LIN {X 0.159,Y -655.159,Z 842.614,A 0.000,B 0.000,C 90.000,E1 326.580} C_DIS
LIN {X 0.166,Y -657.931,Z 842.609,A 0.000,B 0.000,C 90.000,E1 325.595} C_DIS
LIN {X 0.218,Y -660.579,Z 842.604,A 0.000,B 0.000,C 90.000,E1 324.609} C_DIS
LIN {X -0.133,Y -663.447,Z 842.597,A 0.000,B 0.000,C 90.000,E1 323.417} C_DIS
LIN {X -0.112,Y -664.973,Z 842.593,A 0.000,B 0.000,C 90.000,E1 322.683} C_DIS
LIN {X 0.021,Y -666.876,Z 842.587,A 0.000,B 0.000,C 90.000,E1 321.698} C_DIS
LIN {X 0.058,Y -668.914,Z 842.581,A 0.000,B 0.000,C 90.000,E1 320.481} C_DIS
LIN {X -0.293,Y -670.706,Z 842.574,A 0.000,B 0.000,C 90.000,E1 319.299} C_DIS
LIN {X 0.364,Y -673.373,Z 842.563,A 0.000,B 0.000,C 90.000,E1 317.310} C_DIS
LIN {X -0.033,Y -674.352,Z 842.559,A 0.000,B 0.000,C 90.000,E1 316.620} C_DIS
LIN {X 0.016,Y -675.024,Z 842.556,A 0.000,B 0.000,C 90.000,E1 316.134} C_DIS
LIN {X 0.071,Y -675.502,Z 842.554,A 0.000,B 0.000,C 90.000,E1 315.648} C_DIS
LIN {X 0.131,Y -676.141,Z 842.551,A 0.000,B 0.000,C 90.000,E1 315.162} C_DIS
LIN {X 0.331,Y -677.702,Z 842.543,A 0.000,B 0.000,C 90.000,E1 313.704} C_DIS
LIN {X 0.049,Y -678.975,Z 842.536,A 0.000,B 0.000,C 90.000,E1 312.528} C_DIS
LIN {X 0.331,Y -680.489,Z 842.528,A 0.000,B 0.000,C 90.000,E1 311.067} C_DIS
LIN {X 0.196,Y -681.842,Z 842.520,A 0.000,B 0.000,C 90.000,E1 309.644} C_DIS
LIN {X -0.311,Y -683.305,Z 842.511,A 0.000,B 0.000,C 90.000,E1 308.016} C_DIS
LIN {X -0.286,Y -684.517,Z 842.503,A 0.000,B 0.000,C 90.000,E1 306.583} C_DIS
LIN {X 0.318,Y -685.661,Z 842.495,A 0.000,B 0.000,C 90.000,E1 305.105} C_DIS
LIN {X 0.359,Y -686.472,Z 842.489,A 0.000,B 0.000,C 90.000,E1 303.913} C_DIS
LIN {X -0.135,Y -687.817,Z 842.478,A 0.000,B 0.000,C 90.000,E1 302.054} C_DIS
LIN {X 0.207,Y -689.207,Z 842.468,A 0.000,B 0.000,C 90.000,E1 300.129} C_DIS
LIN {X 0.017,Y -690.515,Z 842.458,A 0.000,B 0.000,C 90.000,E1 298.487} C_DIS
LIN {X -0.095,Y -691.710,Z 842.450,A 0.000,B 0.000,C 90.000,E1 297.078} C_DIS
LIN {X 0.068,Y -693.228,Z 842.441,A 0.000,B 0.000,C 90.000,E1 295.412} C_DIS
LIN {X 0.137,Y -694.043,Z 842.436,A 0.000,B 0.000,C 90.000,E1 294.463} C_DIS
LIN {X -0.037,Y -694.284,Z 842.432,A 0.000,B 0.000,C 90.000,E1 293.770} C_DIS
LIN {X 0.182,Y -693.984,Z 842.430,A 0.000,B 0.000,C 90.000,E1 293.281} C_DIS
LIN {X -0.211,Y -693.555,Z 842.428,A 0.000,B 0.000,C 90.000,E1 293.078} C_DIS
LIN {X 0.125,Y -691.002,Z 842.425,A 0.000,B 0.000,C 90.000,E1 292.461} C_DIS
LIN {X 0.242,Y -690.176,Z 842.424,A 0.000,B 0.000,C 90.000,E1 292.333} C_DIS
LIN {X 0.358,Y -688.960,Z 842.424,A 0.000,B 0.000,C 90.000,E1 292.206} C_DIS
LIN {X -0.397,Y -683.079,Z 842.421,A 0.000,B 0.000,C 90.000,E1 291.844} C_DIS
LIN {X -0.059,Y -681.119,Z 842.421,A 0.000,B 0.000,C 90.000,E1 291.716} C_DIS
LIN {X -0.296,Y -671.354,Z 842.419,A 0.000,B 0.000,C 90.000,E1 291.408} C_DIS
LIN {X 0.171,Y -664.788,Z 842.418,A 0.000,B 0.000,C 90.000,E1 291.227} C_DIS
LIN {X -0.028,Y -654.109,Z 842.417,A 0.000,B 0.000,C 90.000,E1 291.046} C_DIS
LIN {X -0.109,Y -648.329,Z 842.416,A 0.000,B 0.000,C 90.000,E1 290.918} C_DIS
LIN {X -0.062,Y -642.259,Z 842.415,A 0.000,B 0.000,C 90.000,E1 290.737} C_DIS
LIN {X -0.135,Y -636.875,Z 842.414,A 0.000,B 0.000,C 90.000,E1 290.536} C_DIS
LIN {X -0.105,Y -634.934,Z 842.414,A 0.000,B 0.000,C 90.000,E1 290.429} C_DIS
LIN {X -0.127,Y -632.025,Z 842.412,A 0.000,B 0.000,C 90.000,E1 290.248} C_DIS
LIN {X -0.160,Y -631.973,Z 842.412,A 0.000,B 0.000,C 90.000,E1 290.248} C_DIS
LIN {X -0.137,Y -631.192,Z 842.412,A 0.000,B 0.000,C 90.000,E1 290.120} C_DIS
LIN {X -0.180,Y -631.170,Z 842.412,A 0.000,B 0.000,C 90.000,E1 290.120} C_DIS
LIN {X -0.162,Y -631.443,Z 842.410,A 0.000,B 0.000,C 90.000,E1 289.885} C_DIS
LIN {X -0.156,Y -631.746,Z 842.410,A 0.000,B 0.000,C 90.000,E1 289.758} C_DIS
LIN {X 0.257,Y -633.950,Z 842.407,A 0.000,B 0.000,C 90.000,E1 289.214} C_DIS
LIN {X -0.086,Y -638.971,Z 842.402,A 0.000,B 0.000,C 90.000,E1 288.362} C_DIS
LIN {X -0.231,Y -641.589,Z 842.399,A 0.000,B 0.000,C 90.000,E1 287.873} C_DIS
LIN {X 0.090,Y -644.996,Z 842.395,A 0.000,B 0.000,C 90.000,E1 287.094} C_DIS
LIN {X -0.211,Y -647.076,Z 842.392,A 0.000,B 0.000,C 90.000,E1 286.622} C_DIS
LIN {X 0.168,Y -649.848,Z 842.388,A 0.000,B 0.000,C 90.000,E1 285.843} C_DIS
LIN {X -0.228,Y -652.100,Z 842.384,A 0.000,B 0.000,C 90.000,E1 285.134} C_DIS
LIN {X 0.319,Y -653.323,Z 842.381,A 0.000,B 0.000,C 90.000,E1 284.592} C_DIS
LIN {X -0.044,Y -654.775,Z 842.377,A 0.000,B 0.000,C 90.000,E1 283.883} C_DIS
LIN {X -0.278,Y -655.578,Z 842.374,A 0.000,B 0.000,C 90.000,E1 283.411} C_DIS
LIN {X 0.017,Y -656.130,Z 842.370,A 0.000,B 0.000,C 90.000,E1 282.647} C_DIS
LIN {X -0.211,Y -656.299,Z 842.368,A 0.000,B 0.000,C 90.000,E1 282.175} C_DIS
LIN {X 0.070,Y -656.221,Z 842.365,A 0.000,B 0.000,C 90.000,E1 281.658} C_DIS
LIN {X -0.158,Y -655.977,Z 842.362,A 0.000,B 0.000,C 90.000,E1 281.186} C_DIS
LIN {X 0.016,Y -655.114,Z 842.358,A 0.000,B 0.000,C 90.000,E1 280.433} C_DIS
LIN {X -0.222,Y -654.223,Z 842.355,A 0.000,B 0.000,C 90.000,E1 279.962} C_DIS
LIN {X 0.064,Y -653.145,Z 842.353,A 0.000,B 0.000,C 90.000,E1 279.443} C_DIS
LIN {X -0.193,Y -651.664,Z 842.350,A 0.000,B 0.000,C 90.000,E1 278.973} C_DIS
LIN {X 0.080,Y -649.679,Z 842.347,A 0.000,B 0.000,C 90.000,E1 278.454} C_DIS
LIN {X 0.312,Y -646.763,Z 842.344,A 0.000,B 0.000,C 90.000,E1 277.814} C_DIS
LIN {X -0.210,Y -643.271,Z 842.340,A 0.000,B 0.000,C 90.000,E1 277.239} C_DIS
LIN {X 0.133,Y -640.882,Z 842.338,A 0.000,B 0.000,C 90.000,E1 276.834} C_DIS
LIN {X -0.119,Y -638.988,Z 842.337,A 0.000,B 0.000,C 90.000,E1 276.606} C_DIS
LIN {X 0.072,Y -634.956,Z 842.334,A 0.000,B 0.000,C 90.000,E1 276.087} C_DIS
LIN {X -0.092,Y -631.561,Z 842.332,A 0.000,B 0.000,C 90.000,E1 275.739} C_DIS
LIN {X -0.193,Y -630.344,Z 842.331,A 0.000,B 0.000,C 90.000,E1 275.625} C_DIS
LIN {X -0.178,Y -625.082,Z 842.329,A 0.000,B 0.000,C 90.000,E1 275.163} C_DIS
LIN {X -0.078,Y -623.753,Z 842.328,A 0.000,B 0.000,C 90.000,E1 275.049} C_DIS
LIN {X -0.272,Y -617.463,Z 842.326,A 0.000,B 0.000,C 90.000,E1 274.645} C_DIS
LIN {X -0.035,Y -611.108,Z 842.324,A 0.000,B 0.000,C 90.000,E1 274.245} C_DIS
LIN {X 0.029,Y -604.288,Z 842.322,A 0.000,B 0.000,C 90.000,E1 273.898} C_DIS
LIN {X -0.269,Y -597.399,Z 842.320,A 0.000,B 0.000,C 90.000,E1 273.612} C_DIS
LIN {X -0.131,Y -591.984,Z 842.319,A 0.000,B 0.000,C 90.000,E1 273.383} C_DIS
LIN {X 0.225,Y -584.869,Z 842.317,A 0.000,B 0.000,C 90.000,E1 273.094} C_DIS
LIN {X -0.174,Y -578.917,Z 842.317,A 0.000,B 0.000,C 90.000,E1 272.980} C_DIS
LIN {X -0.269,Y -572.255,Z 842.316,A 0.000,B 0.000,C 90.000,E1 272.865} C_DIS
LIN {X 0.167,Y -564.435,Z 842.315,A 0.000,B 0.000,C 90.000,E1 272.751} C_DIS
LIN {X 0.112,Y -560.003,Z 842.315,A 0.000,B 0.000,C 90.000,E1 272.751} C_DIS
LIN {X -0.196,Y -554.623,Z 842.315,A 0.000,B 0.000,C 90.000,E1 272.751} C_DIS
LIN {X 0.215,Y -553.395,Z 842.315,A 0.000,B 0.000,C 90.000,E1 272.694} C_DIS
LIN {X 0.227,Y -550.457,Z 842.315,A 0.000,B 0.000,C 90.000,E1 272.579} C_DIS
LIN {X 0.187,Y -550.405,Z 842.315,A 0.000,B 0.000,C 90.000,E1 272.579} C_DIS
LIN {X 0.172,Y -549.400,Z 842.314,A 0.000,B 0.000,C 90.000,E1 272.407} C_DIS
LIN {X 0.209,Y -548.528,Z 842.312,A 0.000,B 0.000,C 90.000,E1 272.121} C_DIS
LIN {X -0.222,Y -547.535,Z 842.309,A 0.000,B 0.000,C 90.000,E1 271.604} C_DIS
LIN {X 0.004,Y -546.052,Z 842.301,A 0.000,B 0.000,C 90.000,E1 270.172} C_DIS
LIN {X -0.267,Y -544.563,Z 842.290,A 0.000,B 0.000,C 90.000,E1 268.224} C_DIS
LIN {X -0.055,Y -543.574,Z 842.282,A 0.000,B 0.000,C 90.000,E1 266.788} C_DIS
LIN {X 0.111,Y -542.607,Z 842.274,A 0.000,B 0.000,C 90.000,E1 265.355} C_DIS
LIN {X -0.193,Y -541.693,Z 842.266,A 0.000,B 0.000,C 90.000,E1 263.970} C_DIS
LIN {X -0.105,Y -541.008,Z 842.262,A 0.000,B 0.000,C 90.000,E1 263.109} C_DIS
LIN {X 0.165,Y -539.463,Z 842.252,A 0.000,B 0.000,C 90.000,E1 261.376} C_DIS
LIN {X -0.116,Y -538.157,Z 842.244,A 0.000,B 0.000,C 90.000,E1 259.982} C_DIS
LIN {X -0.196,Y -536.114,Z 842.233,A 0.000,B 0.000,C 90.000,E1 257.993} C_DIS
LIN {X 0.083,Y -534.647,Z 842.225,A 0.000,B 0.000,C 90.000,E1 256.533} C_DIS
LIN {X 0.150,Y -532.322,Z 842.214,A 0.000,B 0.000,C 90.000,E1 254.519} C_DIS
LIN {X 0.279,Y -530.289,Z 842.205,A 0.000,B 0.000,C 90.000,E1 252.779} C_DIS
LIN {X 0.175,Y -528.869,Z 842.198,A 0.000,B 0.000,C 90.000,E1 251.638} C_DIS
LIN {X 0.220,Y -527.017,Z 842.190,A 0.000,B 0.000,C 90.000,E1 250.188} C_DIS
LIN {X 0.085,Y -524.639,Z 842.180,A 0.000,B 0.000,C 90.000,E1 248.465} C_DIS
LIN {X -0.103,Y -522.166,Z 842.171,A 0.000,B 0.000,C 90.000,E1 246.741} C_DIS
LIN {X 0.245,Y -520.450,Z 842.164,A 0.000,B 0.000,C 90.000,E1 245.537} C_DIS
LIN {X -0.089,Y -517.597,Z 842.155,A 0.000,B 0.000,C 90.000,E1 243.819} C_DIS
LIN {X 0.206,Y -514.481,Z 842.145,A 0.000,B 0.000,C 90.000,E1 242.025} C_DIS
LIN {X 0.214,Y -511.357,Z 842.135,A 0.000,B 0.000,C 90.000,E1 240.255} C_DIS
LIN {X 0.036,Y -507.500,Z 842.123,A 0.000,B 0.000,C 90.000,E1 238.201} C_DIS
LIN {X -0.229,Y -505.155,Z 842.117,A 0.000,B 0.000,C 90.000,E1 237.041} C_DIS
LIN {X 0.171,Y -502.596,Z 842.110,A 0.000,B 0.000,C 90.000,E1 235.801} C_DIS
LIN {X 0.118,Y -499.881,Z 842.104,A 0.000,B 0.000,C 90.000,E1 234.609} C_DIS
LIN {X 0.317,Y -494.874,Z 842.092,A 0.000,B 0.000,C 90.000,E1 232.477} C_DIS
LIN {X -0.093,Y -491.372,Z 842.083,A 0.000,B 0.000,C 90.000,E1 231.009} C_DIS
LIN {X 0.120,Y -487.860,Z 842.075,A 0.000,B 0.000,C 90.000,E1 229.461} C_DIS
LIN {X 0.069,Y -485.043,Z 842.068,A 0.000,B 0.000,C 90.000,E1 228.243} C_DIS
LIN {X -0.191,Y -479.580,Z 842.054,A 0.000,B 0.000,C 90.000,E1 225.810} C_DIS
LIN {X -0.272,Y -476.245,Z 842.046,A 0.000,B 0.000,C 90.000,E1 224.271} C_DIS
LIN {X -0.206,Y -471.460,Z 842.034,A 0.000,B 0.000,C 90.000,E1 222.081} C_DIS
LIN {X 0.240,Y -468.092,Z 842.025,A 0.000,B 0.000,C 90.000,E1 220.458} C_DIS
LIN {X 0.062,Y -464.269,Z 842.014,A 0.000,B 0.000,C 90.000,E1 218.588} C_DIS
LIN {X -0.020,Y -459.674,Z 842.002,A 0.000,B 0.000,C 90.000,E1 216.377} C_DIS
LIN {X -0.129,Y -454.179,Z 841.988,A 0.000,B 0.000,C 90.000,E1 213.833} C_DIS
LIN {X 0.137,Y -449.359,Z 841.975,A 0.000,B 0.000,C 90.000,E1 211.544} C_DIS
LIN {X 0.108,Y -443.953,Z 841.961,A 0.000,B 0.000,C 90.000,E1 208.949} C_DIS
LIN {X 0.064,Y -441.992,Z 841.956,A 0.000,B 0.000,C 90.000,E1 207.975} C_DIS
LIN {X -0.098,Y -438.073,Z 841.945,A 0.000,B 0.000,C 90.000,E1 206.027} C_DIS
LIN {X -0.171,Y -434.659,Z 841.935,A 0.000,B 0.000,C 90.000,E1 204.387} C_DIS
LIN {X -0.083,Y -431.285,Z 841.926,A 0.000,B 0.000,C 90.000,E1 202.717} C_DIS
LIN {X -0.055,Y -428.085,Z 841.917,A 0.000,B 0.000,C 90.000,E1 201.046} C_DIS
LIN {X -0.245,Y -424.786,Z 841.908,A 0.000,B 0.000,C 90.000,E1 199.396} C_DIS
LIN {X 0.114,Y -422.197,Z 841.900,A 0.000,B 0.000,C 90.000,E1 198.000} C_DIS
LIN {X -0.127,Y -417.669,Z 841.887,A 0.000,B 0.000,C 90.000,E1 195.662} C_DIS
LIN {X -0.131,Y -414.950,Z 841.879,A 0.000,B 0.000,C 90.000,E1 194.300} C_DIS
LIN {X -0.114,Y -410.810,Z 841.868,A 0.000,B 0.000,C 90.000,E1 192.243} C_DIS
LIN {X 0.123,Y -406.864,Z 841.857,A 0.000,B 0.000,C 90.000,E1 190.141} C_DIS
LIN {X 0.188,Y -402.908,Z 841.845,A 0.000,B 0.000,C 90.000,E1 188.049} C_DIS
LIN {X 0.004,Y -397.565,Z 841.829,A 0.000,B 0.000,C 90.000,E1 185.277} C_DIS
LIN {X -0.130,Y -392.477,Z 841.812,A 0.000,B 0.000,C 90.000,E1 182.121} C_DIS
LIN {X -0.169,Y -387.666,Z 841.792,A 0.000,B 0.000,C 90.000,E1 178.568} C_DIS
LIN {X -0.155,Y -383.843,Z 841.776,A 0.000,B 0.000,C 90.000,E1 175.698} C_DIS
LIN {X 0.114,Y -381.571,Z 841.766,A 0.000,B 0.000,C 90.000,E1 173.856} C_DIS
LIN {X 0.035,Y -378.185,Z 841.750,A 0.000,B 0.000,C 90.000,E1 170.971} C_DIS
LIN {X -0.139,Y -375.977,Z 841.738,A 0.000,B 0.000,C 90.000,E1 168.814} C_DIS
LIN {X 0.047,Y -373.886,Z 841.724,A 0.000,B 0.000,C 90.000,E1 166.228} C_DIS
LIN {X 0.032,Y -372.437,Z 841.711,A 0.000,B 0.000,C 90.000,E1 164.031} C_DIS
LIN {X 0.120,Y -371.897,Z 841.701,A 0.000,B 0.000,C 90.000,E1 162.181} C_DIS
LIN {X 0.019,Y -371.980,Z 841.695,A 0.000,B 0.000,C 90.000,E1 161.094} C_DIS
LIN {X -0.082,Y -372.367,Z 841.689,A 0.000,B 0.000,C 90.000,E1 160.007} C_DIS
LIN {X -0.052,Y -373.342,Z 841.683,A 0.000,B 0.000,C 90.000,E1 158.901} C_DIS
LIN {X 0.021,Y -374.351,Z 841.679,A 0.000,B 0.000,C 90.000,E1 158.156} C_DIS
LIN {X 0.105,Y -375.655,Z 841.675,A 0.000,B 0.000,C 90.000,E1 157.411} C_DIS
LIN {X 0.092,Y -375.914,Z 841.674,A 0.000,B 0.000,C 90.000,E1 157.230} C_DIS
LIN {X -0.118,Y -377.023,Z 841.671,A 0.000,B 0.000,C 90.000,E1 156.847} C_DIS
LIN {X -0.142,Y -377.825,Z 841.669,A 0.000,B 0.000,C 90.000,E1 156.485} C_DIS
LIN {X -0.013,Y -379.178,Z 841.667,A 0.000,B 0.000,C 90.000,E1 156.102} C_DIS
LIN {X 0.118,Y -381.011,Z 841.664,A 0.000,B 0.000,C 90.000,E1 155.537} C_DIS
LIN {X -0.034,Y -383.713,Z 841.662,A 0.000,B 0.000,C 90.000,E1 155.101} C_DIS
LIN {X 0.161,Y -387.096,Z 841.659,A 0.000,B 0.000,C 90.000,E1 154.588} C_DIS
LIN {X -0.131,Y -389.702,Z 841.657,A 0.000,B 0.000,C 90.000,E1 154.332} C_DIS
LIN {X 0.083,Y -396.236,Z 841.655,A 0.000,B 0.000,C 90.000,E1 153.845} C_DIS
LIN {X -0.151,Y -398.235,Z 841.654,A 0.000,B 0.000,C 90.000,E1 153.768} C_DIS
LIN {X 0.052,Y -405.159,Z 841.653,A 0.000,B 0.000,C 90.000,E1 153.435} C_DIS
LIN {X -0.082,Y -409.417,Z 841.652,A 0.000,B 0.000,C 90.000,E1 153.307} C_DIS
LIN {X -0.087,Y -415.622,Z 841.650,A 0.000,B 0.000,C 90.000,E1 153.050} C_DIS
LIN {X 0.074,Y -420.584,Z 841.649,A 0.000,B 0.000,C 90.000,E1 152.794} C_DIS
LIN {X -0.239,Y -425.539,Z 841.648,A 0.000,B 0.000,C 90.000,E1 152.615} C_DIS
LIN {X -0.107,Y -433.645,Z 841.645,A 0.000,B 0.000,C 90.000,E1 152.153} C_DIS
LIN {X -0.093,Y -438.451,Z 841.644,A 0.000,B 0.000,C 90.000,E1 151.847} C_DIS
LIN {X 0.044,Y -447.924,Z 841.640,A 0.000,B 0.000,C 90.000,E1 151.179} C_DIS
LIN {X -0.059,Y -455.453,Z 841.637,A 0.000,B 0.000,C 90.000,E1 150.589} C_DIS
LIN {X -0.025,Y -460.039,Z 841.635,A 0.000,B 0.000,C 90.000,E1 150.205} C_DIS
LIN {X 0.114,Y -464.314,Z 841.632,A 0.000,B 0.000,C 90.000,E1 149.793} C_DIS
LIN {X 0.193,Y -474.143,Z 841.627,A 0.000,B 0.000,C 90.000,E1 148.791} C_DIS
LIN {X 0.122,Y -482.141,Z 841.622,A 0.000,B 0.000,C 90.000,E1 147.946} C_DIS
LIN {X -0.154,Y -485.975,Z 841.620,A 0.000,B 0.000,C 90.000,E1 147.533} C_DIS
LIN {X 0.123,Y -489.732,Z 841.617,A 0.000,B 0.000,C 90.000,E1 147.041} C_DIS
LIN {X -0.142,Y -496.900,Z 841.612,A 0.000,B 0.000,C 90.000,E1 146.167} C_DIS
LIN {X 0.023,Y -501.139,Z 841.609,A 0.000,B 0.000,C 90.000,E1 145.548} C_DIS
LIN {X -0.026,Y -508.826,Z 841.602,A 0.000,B 0.000,C 90.000,E1 144.356} C_DIS
LIN {X -0.068,Y -516.064,Z 841.595,A 0.000,B 0.000,C 90.000,E1 143.176} C_DIS
LIN {X 0.058,Y -524.892,Z 841.587,A 0.000,B 0.000,C 90.000,E1 141.698} C_DIS
LIN {X -0.323,Y -532.304,Z 841.580,A 0.000,B 0.000,C 90.000,E1 140.436} C_DIS
LIN {X 0.165,Y -539.318,Z 841.573,A 0.000,B 0.000,C 90.000,E1 139.094} C_DIS
LIN {X -0.234,Y -545.312,Z 841.567,A 0.000,B 0.000,C 90.000,E1 138.000} C_DIS
LIN {X -0.129,Y -552.657,Z 841.559,A 0.000,B 0.000,C 90.000,E1 136.581} C_DIS
LIN {X 0.002,Y -557.212,Z 841.554,A 0.000,B 0.000,C 90.000,E1 135.729} C_DIS
LIN {X -0.317,Y -563.468,Z 841.547,A 0.000,B 0.000,C 90.000,E1 134.514} C_DIS
LIN {X 0.322,Y -567.391,Z 841.543,A 0.000,B 0.000,C 90.000,E1 133.623} C_DIS
LIN {X -0.111,Y -574.470,Z 841.534,A 0.000,B 0.000,C 90.000,E1 132.162} C_DIS
LIN {X -0.022,Y -579.331,Z 841.528,A 0.000,B 0.000,C 90.000,E1 131.067} C_DIS
LIN {X 0.018,Y -582.730,Z 841.524,A 0.000,B 0.000,C 90.000,E1 130.253} C_DIS
LIN {X -0.172,Y -587.215,Z 841.518,A 0.000,B 0.000,C 90.000,E1 129.197} C_DIS
LIN {X -0.050,Y -590.223,Z 841.513,A 0.000,B 0.000,C 90.000,E1 128.382} C_DIS
LIN {X 0.101,Y -592.966,Z 841.509,A 0.000,B 0.000,C 90.000,E1 127.569} C_DIS
LIN {X 0.174,Y -594.649,Z 841.506,A 0.000,B 0.000,C 90.000,E1 127.030} C_DIS
LIN {X -0.005,Y -598.282,Z 841.499,A 0.000,B 0.000,C 90.000,E1 125.724} C_DIS
LIN {X -0.133,Y -600.105,Z 841.494,A 0.000,B 0.000,C 90.000,E1 124.945} C_DIS
LIN {X 0.253,Y -601.667,Z 841.490,A 0.000,B 0.000,C 90.000,E1 124.119} C_DIS
LIN {X 0.069,Y -603.450,Z 841.484,A 0.000,B 0.000,C 90.000,E1 123.086} C_DIS
LIN {X -0.095,Y -604.889,Z 841.478,A 0.000,B 0.000,C 90.000,E1 122.054} C_DIS
LIN {X 0.205,Y -606.445,Z 841.471,A 0.000,B 0.000,C 90.000,E1 120.718} C_DIS
LIN {X 0.035,Y -607.113,Z 841.466,A 0.000,B 0.000,C 90.000,E1 119.951} C_DIS
LIN {X 0.131,Y -607.518,Z 841.461,A 0.000,B 0.000,C 90.000,E1 118.899} C_DIS
LIN {X 0.275,Y -607.600,Z 841.456,A 0.000,B 0.000,C 90.000,E1 118.103} C_DIS
LIN {X 0.134,Y -607.420,Z 841.452,A 0.000,B 0.000,C 90.000,E1 117.334} C_DIS
LIN {X -0.054,Y -606.589,Z 841.446,A 0.000,B 0.000,C 90.000,E1 116.309} C_DIS
LIN {X -0.203,Y -605.672,Z 841.442,A 0.000,B 0.000,C 90.000,E1 115.540} C_DIS
LIN {X -0.310,Y -604.992,Z 841.439,A 0.000,B 0.000,C 90.000,E1 115.027} C_DIS
LIN {X 0.127,Y -604.027,Z 841.436,A 0.000,B 0.000,C 90.000,E1 114.463} C_DIS
LIN {X 0.068,Y -603.460,Z 841.435,A 0.000,B 0.000,C 90.000,E1 114.207} C_DIS
LIN {X 0.118,Y -600.622,Z 841.429,A 0.000,B 0.000,C 90.000,E1 113.153} C_DIS
LIN {X -0.070,Y -598.001,Z 841.425,A 0.000,B 0.000,C 90.000,E1 112.514} C_DIS
LIN {X 0.129,Y -594.958,Z 841.423,A 0.000,B 0.000,C 90.000,E1 112.099} C_DIS
LIN {X 0.080,Y -593.465,Z 841.422,A 0.000,B 0.000,C 90.000,E1 111.897} C_DIS
LIN {X -0.213,Y -589.284,Z 841.420,A 0.000,B 0.000,C 90.000,E1 111.535} C_DIS
LIN {X -0.187,Y -587.690,Z 841.419,A 0.000,B 0.000,C 90.000,E1 111.408} C_DIS
LIN {X 0.030,Y -580.830,Z 841.417,A 0.000,B 0.000,C 90.000,E1 110.972} C_DIS
LIN {X -0.207,Y -574.192,Z 841.415,A 0.000,B 0.000,C 90.000,E1 110.663} C_DIS
LIN {X -0.116,Y -570.988,Z 841.414,A 0.000,B 0.000,C 90.000,E1 110.482} C_DIS
LIN {X 0.069,Y -567.730,Z 841.413,A 0.000,B 0.000,C 90.000,E1 110.248} C_DIS
LIN {X -0.291,Y -565.914,Z 841.412,A 0.000,B 0.000,C 90.000,E1 110.120} C_DIS
LIN {X -0.221,Y -565.462,Z 841.411,A 0.000,B 0.000,C 90.000,E1 110.066} C_DIS
LIN {X -0.259,Y -565.434,Z 841.411,A 0.000,B 0.000,C 90.000,E1 110.066} C_DIS
LIN {X -0.044,Y -564.702,Z 841.410,A 0.000,B 0.000,C 90.000,E1 109.758} C_DIS
LIN {X 0.179,Y -563.228,Z 841.407,A 0.000,B 0.000,C 90.000,E1 109.322} C_DIS
LIN {X 0.209,Y -562.488,Z 841.405,A 0.000,B 0.000,C 90.000,E1 108.906} C_DIS
LIN {X 0.127,Y -561.855,Z 841.402,A 0.000,B 0.000,C 90.000,E1 108.362} C_DIS
LIN {X 0.088,Y -561.309,Z 841.394,A 0.000,B 0.000,C 90.000,E1 106.985} C_DIS
LIN {X -0.189,Y -562.582,Z 841.370,A 0.000,B 0.000,C 90.000,E1 102.591} C_DIS
LIN {X 0.145,Y -564.202,Z 841.356,A 0.000,B 0.000,C 90.000,E1 100.074} C_DIS
LIN {X 0.224,Y -565.193,Z 841.348,A 0.000,B 0.000,C 90.000,E1 98.690} C_DIS
LIN {X -0.058,Y -566.273,Z 841.339,A 0.000,B 0.000,C 90.000,E1 97.068} C_DIS
LIN {X 0.229,Y -567.189,Z 841.330,A 0.000,B 0.000,C 90.000,E1 95.391} C_DIS
LIN {X 0.151,Y -567.655,Z 841.324,A 0.000,B 0.000,C 90.000,E1 94.302} C_DIS
LIN {X 0.237,Y -568.193,Z 841.316,A 0.000,B 0.000,C 90.000,E1 92.922} C_DIS
LIN {X -0.149,Y -568.671,Z 841.307,A 0.000,B 0.000,C 90.000,E1 91.318} C_DIS
LIN {X -0.091,Y -569.052,Z 841.300,A 0.000,B 0.000,C 90.000,E1 89.943} C_DIS
LIN {X 0.097,Y -569.470,Z 841.291,A 0.000,B 0.000,C 90.000,E1 88.282} C_DIS
LIN {X -0.235,Y -569.771,Z 841.281,A 0.000,B 0.000,C 90.000,E1 86.674} C_DIS
LIN {X 0.018,Y -570.053,Z 841.272,A 0.000,B 0.000,C 90.000,E1 85.008} C_DIS
LIN {X 0.147,Y -570.332,Z 841.265,A 0.000,B 0.000,C 90.000,E1 83.628} C_DIS
LIN {X 0.248,Y -570.868,Z 841.253,A 0.000,B 0.000,C 90.000,E1 81.432} C_DIS
LIN {X 0.071,Y -571.619,Z 841.239,A 0.000,B 0.000,C 90.000,E1 78.993} C_DIS
LIN {X -0.086,Y -572.083,Z 841.231,A 0.000,B 0.000,C 90.000,E1 77.645} C_DIS
LIN {X 0.094,Y -572.516,Z 841.222,A 0.000,B 0.000,C 90.000,E1 75.992} C_DIS
LIN {X 0.094,Y -572.811,Z 841.215,A 0.000,B 0.000,C 90.000,E1 74.629} C_DIS
LIN {X -0.108,Y -572.961,Z 841.206,A 0.000,B 0.000,C 90.000,E1 73.015} C_DIS
LIN {X 0.041,Y -572.948,Z 841.195,A 0.000,B 0.000,C 90.000,E1 71.094} C_DIS
LIN {X -0.177,Y -572.820,Z 841.184,A 0.000,B 0.000,C 90.000,E1 69.209} C_DIS
LIN {X 0.015,Y -572.524,Z 841.174,A 0.000,B 0.000,C 90.000,E1 67.283} C_DIS
LIN {X 0.010,Y -572.215,Z 841.166,A 0.000,B 0.000,C 90.000,E1 65.921} C_DIS
LIN {X 0.223,Y -571.700,Z 841.159,A 0.000,B 0.000,C 90.000,E1 64.537} C_DIS
LIN {X -0.095,Y -571.173,Z 841.151,A 0.000,B 0.000,C 90.000,E1 63.204} C_DIS
LIN {X -0.167,Y -570.628,Z 841.144,A 0.000,B 0.000,C 90.000,E1 61.847} C_DIS
LIN {X 0.094,Y -570.203,Z 841.139,A 0.000,B 0.000,C 90.000,E1 61.001} C_DIS
LIN {X -0.148,Y -569.595,Z 841.134,A 0.000,B 0.000,C 90.000,E1 60.205} C_DIS
LIN {X -0.215,Y -569.162,Z 841.131,A 0.000,B 0.000,C 90.000,E1 59.665} C_DIS
LIN {X 0.134,Y -568.048,Z 841.125,A 0.000,B 0.000,C 90.000,E1 58.535} C_DIS
LIN {X -0.019,Y -566.781,Z 841.119,A 0.000,B 0.000,C 90.000,E1 57.454} C_DIS
LIN {X 0.120,Y -565.356,Z 841.113,A 0.000,B 0.000,C 90.000,E1 56.342} C_DIS
LIN {X 0.135,Y -564.112,Z 841.109,A 0.000,B 0.000,C 90.000,E1 55.515} C_DIS
LIN {X 0.133,Y -562.749,Z 841.104,A 0.000,B 0.000,C 90.000,E1 54.689} C_DIS
LIN {X -0.243,Y -560.619,Z 841.098,A 0.000,B 0.000,C 90.000,E1 53.623} C_DIS
LIN {X 0.136,Y -558.172,Z 841.092,A 0.000,B 0.000,C 90.000,E1 52.477} C_DIS
LIN {X 0.310,Y -556.839,Z 841.089,A 0.000,B 0.000,C 90.000,E1 51.904} C_DIS
LIN {X 0.037,Y -555.391,Z 841.086,A 0.000,B 0.000,C 90.000,E1 51.376} C_DIS
LIN {X -0.170,Y -552.947,Z 841.081,A 0.000,B 0.000,C 90.000,E1 50.561} C_DIS
LIN {X 0.020,Y -550.189,Z 841.076,A 0.000,B 0.000,C 90.000,E1 49.703} C_DIS
LIN {X 0.065,Y -548.188,Z 841.073,A 0.000,B 0.000,C 90.000,E1 49.138} C_DIS
LIN {X -0.220,Y -544.804,Z 841.068,A 0.000,B 0.000,C 90.000,E1 48.324} C_DIS
LIN {X -0.010,Y -541.737,Z 841.064,A 0.000,B 0.000,C 90.000,E1 47.595} C_DIS
LIN {X -0.192,Y -538.336,Z 841.061,A 0.000,B 0.000,C 90.000,E1 46.905} C_DIS
LIN {X -0.011,Y -536.205,Z 841.058,A 0.000,B 0.000,C 90.000,E1 46.458} C_DIS
LIN {X 0.120,Y -532.160,Z 841.054,A 0.000,B 0.000,C 90.000,E1 45.729} C_DIS
LIN {X 0.213,Y -527.579,Z 841.050,A 0.000,B 0.000,C 90.000,E1 45.000} C_DIS
LIN {X -0.048,Y -524.676,Z 841.048,A 0.000,B 0.000,C 90.000,E1 44.595} C_DIS
LIN {X -0.171,Y -520.460,Z 841.045,A 0.000,B 0.000,C 90.000,E1 44.028} C_DIS
LIN {X 0.112,Y -515.952,Z 841.041,A 0.000,B 0.000,C 90.000,E1 43.419} C_DIS
LIN {X -0.158,Y -512.463,Z 841.039,A 0.000,B 0.000,C 90.000,E1 43.014} C_DIS
LIN {X -0.222,Y -507.489,Z 841.036,A 0.000,B 0.000,C 90.000,E1 42.447} C_DIS
LIN {X 0.104,Y -502.201,Z 841.033,A 0.000,B 0.000,C 90.000,E1 41.838} C_DIS
LIN {X -0.121,Y -498.079,Z 841.030,A 0.000,B 0.000,C 90.000,E1 41.434} C_DIS
LIN {X -0.004,Y -492.388,Z 841.027,A 0.000,B 0.000,C 90.000,E1 40.862} C_DIS
LIN {X 0.000,Y -487.950,Z 841.025,A 0.000,B 0.000,C 90.000,E1 40.458} C_DIS
LIN {X 0.060,Y -480.431,Z 841.021,A 0.000,B 0.000,C 90.000,E1 39.806} C_DIS
LIN {X -0.065,Y -471.194,Z 841.017,A 0.000,B 0.000,C 90.000,E1 39.072} C_DIS
LIN {X 0.048,Y -460.282,Z 841.012,A 0.000,B 0.000,C 90.000,E1 38.222} C_DIS
LIN {X -0.133,Y -450.808,Z 841.008,A 0.000,B 0.000,C 90.000,E1 37.523} C_DIS
LIN {X -0.083,Y -433.679,Z 841.001,A 0.000,B 0.000,C 90.000,E1 36.217} C_DIS
LIN {X 0.186,Y -413.625,Z 840.992,A 0.000,B 0.000,C 90.000,E1 34.532} C_DIS
LIN {X 0.017,Y -403.190,Z 840.987,A 0.000,B 0.000,C 90.000,E1 33.579} C_DIS
LIN {X -0.206,Y -399.048,Z 840.984,A 0.000,B 0.000,C 90.000,E1 33.166} C_DIS
LIN {X -0.075,Y -396.185,Z 840.982,A 0.000,B 0.000,C 90.000,E1 32.752} C_DIS
LIN {X 0.134,Y -394.730,Z 840.981,A 0.000,B 0.000,C 90.000,E1 32.467} C_DIS
LIN {X 0.096,Y -394.702,Z 840.980,A 0.000,B 0.000,C 90.000,E1 32.467} C_DIS
LIN {X -0.093,Y -393.711,Z 840.977,A 0.000,B 0.000,C 90.000,E1 31.799} C_DIS
LIN {X 0.155,Y -390.816,Z 840.968,A 0.000,B 0.000,C 90.000,E1 30.256} C_DIS
LIN {X 0.020,Y -391.511,Z 840.957,A 0.000,B 0.000,C 90.000,E1 28.231} C_DIS
LIN {X 0.193,Y -393.046,Z 840.943,A 0.000,B 0.000,C 90.000,E1 25.720} C_DIS
LIN {X 0.066,Y -394.908,Z 840.929,A 0.000,B 0.000,C 90.000,E1 23.259} C_DIS
LIN {X -0.022,Y -396.671,Z 840.918,A 0.000,B 0.000,C 90.000,E1 21.153} C_DIS
LIN {X -0.117,Y -399.779,Z 840.900,A 0.000,B 0.000,C 90.000,E1 18.000} C_DIS
LIN {X -0.113,Y -402.243,Z 840.888,A 0.000,B 0.000,C 90.000,E1 15.898} C_DIS
LIN {X -0.170,Y -406.598,Z 840.871,A 0.000,B 0.000,C 90.000,E1 12.771} C_DIS
LIN {X 0.163,Y -411.598,Z 840.854,A 0.000,B 0.000,C 90.000,E1 9.613} C_DIS
LIN {X -0.081,Y -415.129,Z 840.842,A 0.000,B 0.000,C 90.000,E1 7.587} C_DIS
LIN {X 0.124,Y -418.790,Z 840.831,A 0.000,B 0.000,C 90.000,E1 5.511} C_DIS
LIN {X -0.004,Y -423.272,Z 840.818,A 0.000,B 0.000,C 90.000,E1 3.154} C_DIS
LIN {X 0.027,Y -428.951,Z 840.803,A 0.000,B 0.000,C 90.000,E1 0.458} C_DIS
LIN {X -0.204,Y -435.126,Z 840.788,A 0.000,B 0.000,C 90.000,E1 357.822} C_DIS
LIN {X -0.004,Y -439.978,Z 840.777,A 0.000,B 0.000,C 90.000,E1 355.812} C_DIS
LIN {X -0.074,Y -447.719,Z 840.760,A 0.000,B 0.000,C 90.000,E1 352.875} C_DIS
LIN {X -0.212,Y -450.066,Z 840.757,A 0.000,B 0.000,C 90.000,E1 352.243} C_DIS
LIN {X 0.047,Y -452.420,Z 840.754,A 0.000,B 0.000,C 90.000,E1 351.724} C_DIS
LIN {X 0.180,Y -453.458,Z 840.753,A 0.000,B 0.000,C 90.000,E1 351.546} C_DIS
LIN {X 0.041,Y -456.808,Z 840.751,A 0.000,B 0.000,C 90.000,E1 351.197} C_DIS
LIN {X 0.198,Y -458.427,Z 840.750,A 0.000,B 0.000,C 90.000,E1 351.027} C_DIS
LIN {X -0.026,Y -460.383,Z 840.750,A 0.000,B 0.000,C 90.000,E1 350.905} C_DIS
LIN {X -0.039,Y -465.736,Z 840.748,A 0.000,B 0.000,C 90.000,E1 350.557} C_DIS
LIN {X -0.025,Y -472.913,Z 840.745,A 0.000,B 0.000,C 90.000,E1 350.151} C_DIS
LIN {X -0.221,Y -480.589,Z 840.743,A 0.000,B 0.000,C 90.000,E1 349.746} C_DIS
LIN {X 0.218,Y -488.689,Z 840.740,A 0.000,B 0.000,C 90.000,E1 349.218} C_DIS
LIN {X 0.213,Y -499.843,Z 840.736,A 0.000,B 0.000,C 90.000,E1 348.522} C_DIS
LIN {X -0.087,Y -509.227,Z 840.733,A 0.000,B 0.000,C 90.000,E1 347.937} C_DIS
LIN {X 0.037,Y -518.569,Z 840.729,A 0.000,B 0.000,C 90.000,E1 347.285} C_DIS
LIN {X -0.126,Y -527.700,Z 840.726,A 0.000,B 0.000,C 90.000,E1 346.645} C_DIS
LIN {X 0.097,Y -533.672,Z 840.723,A 0.000,B 0.000,C 90.000,E1 346.172} C_DIS
LIN {X 0.229,Y -539.588,Z 840.721,A 0.000,B 0.000,C 90.000,E1 345.700} C_DIS
LIN {X 0.187,Y -546.737,Z 840.717,A 0.000,B 0.000,C 90.000,E1 345.117} C_DIS
LIN {X 0.080,Y -553.608,Z 840.714,A 0.000,B 0.000,C 90.000,E1 344.519} C_DIS
LIN {X -0.229,Y -560.338,Z 840.711,A 0.000,B 0.000,C 90.000,E1 343.921} C_DIS
LIN {X -0.046,Y -565.439,Z 840.708,A 0.000,B 0.000,C 90.000,E1 343.378} C_DIS
LIN {X -0.037,Y -570.459,Z 840.705,A 0.000,B 0.000,C 90.000,E1 342.834} C_DIS
LIN {X 0.215,Y -576.424,Z 840.701,A 0.000,B 0.000,C 90.000,E1 342.127} C_DIS
LIN {X -0.238,Y -579.791,Z 840.699,A 0.000,B 0.000,C 90.000,E1 341.764} C_DIS
LIN {X -0.281,Y -584.969,Z 840.695,A 0.000,B 0.000,C 90.000,E1 341.094} C_DIS
LIN {X 0.215,Y -590.949,Z 840.690,A 0.000,B 0.000,C 90.000,E1 340.242} C_DIS
LIN {X 0.222,Y -596.114,Z 840.686,A 0.000,B 0.000,C 90.000,E1 339.444} C_DIS
LIN {X 0.066,Y -601.022,Z 840.682,A 0.000,B 0.000,C 90.000,E1 338.666} C_DIS
LIN {X -0.164,Y -605.655,Z 840.677,A 0.000,B 0.000,C 90.000,E1 337.901} C_DIS
LIN {X -0.336,Y -613.097,Z 840.670,A 0.000,B 0.000,C 90.000,E1 336.613} C_DIS
LIN {X 0.118,Y -618.570,Z 840.664,A 0.000,B 0.000,C 90.000,E1 335.537} C_DIS
LIN {X -0.173,Y -623.739,Z 840.659,A 0.000,B 0.000,C 90.000,E1 334.537} C_DIS
LIN {X -0.141,Y -628.000,Z 840.654,A 0.000,B 0.000,C 90.000,E1 333.640} C_DIS
LIN {X -0.050,Y -632.554,Z 840.648,A 0.000,B 0.000,C 90.000,E1 332.615} C_DIS
LIN {X 0.100,Y -636.814,Z 840.642,A 0.000,B 0.000,C 90.000,E1 331.591} C_DIS
LIN {X 0.109,Y -641.901,Z 840.635,A 0.000,B 0.000,C 90.000,E1 330.333} C_DIS
LIN {X 0.136,Y -645.701,Z 840.630,A 0.000,B 0.000,C 90.000,E1 329.331} C_DIS
LIN {X 0.214,Y -649.213,Z 840.624,A 0.000,B 0.000,C 90.000,E1 328.329} C_DIS
LIN {X -0.128,Y -653.309,Z 840.617,A 0.000,B 0.000,C 90.000,E1 327.120} C_DIS
LIN {X -0.056,Y -655.662,Z 840.613,A 0.000,B 0.000,C 90.000,E1 326.373} C_DIS
LIN {X 0.050,Y -659.037,Z 840.606,A 0.000,B 0.000,C 90.000,E1 325.135} C_DIS
LIN {X 0.014,Y -661.002,Z 840.602,A 0.000,B 0.000,C 90.000,E1 324.402} C_DIS
LIN {X 0.105,Y -663.325,Z 840.597,A 0.000,B 0.000,C 90.000,E1 323.417} C_DIS
LIN {X -0.310,Y -665.368,Z 840.591,A 0.000,B 0.000,C 90.000,E1 322.477} C_DIS
LIN {X 0.238,Y -667.252,Z 840.586,A 0.000,B 0.000,C 90.000,E1 321.457} C_DIS
LIN {X -0.131,Y -668.907,Z 840.581,A 0.000,B 0.000,C 90.000,E1 320.517} C_DIS
LIN {X -0.056,Y -670.753,Z 840.574,A 0.000,B 0.000,C 90.000,E1 319.299} C_DIS
LIN {X -0.347,Y -673.511,Z 840.563,A 0.000,B 0.000,C 90.000,E1 317.391} C_DIS
LIN {X 0.209,Y -674.496,Z 840.559,A 0.000,B 0.000,C 90.000,E1 316.620} C_DIS
LIN {X 0.286,Y -675.394,Z 840.555,A 0.000,B 0.000,C 90.000,E1 315.891} C_DIS
LIN {X -0.071,Y -676.591,Z 840.550,A 0.000,B 0.000,C 90.000,E1 314.960} C_DIS
LIN {X -0.343,Y -678.154,Z 840.542,A 0.000,B 0.000,C 90.000,E1 313.542} C_DIS
LIN {X -0.078,Y -679.667,Z 840.534,A 0.000,B 0.000,C 90.000,E1 312.081} C_DIS
LIN {X 0.180,Y -680.915,Z 840.527,A 0.000,B 0.000,C 90.000,E1 310.862} C_DIS
LIN {X 0.060,Y -682.270,Z 840.519,A 0.000,B 0.000,C 90.000,E1 309.439} C_DIS
LIN {X -0.432,Y -683.713,Z 840.510,A 0.000,B 0.000,C 90.000,E1 307.810} C_DIS
LIN {X -0.395,Y -684.926,Z 840.502,A 0.000,B 0.000,C 90.000,E1 306.377} C_DIS
LIN {X 0.033,Y -685.887,Z 840.495,A 0.000,B 0.000,C 90.000,E1 305.152} C_DIS
LIN {X -0.104,Y -687.025,Z 840.486,A 0.000,B 0.000,C 90.000,E1 303.499} C_DIS
LIN {X -0.215,Y -688.032,Z 840.478,A 0.000,B 0.000,C 90.000,E1 302.084} C_DIS
LIN {X -0.077,Y -689.264,Z 840.469,A 0.000,B 0.000,C 90.000,E1 300.413} C_DIS
LIN {X 0.314,Y -690.735,Z 840.458,A 0.000,B 0.000,C 90.000,E1 298.487} C_DIS
LIN {X 0.207,Y -691.906,Z 840.451,A 0.000,B 0.000,C 90.000,E1 297.078} C_DIS
LIN {X -0.251,Y -693.397,Z 840.441,A 0.000,B 0.000,C 90.000,E1 295.463} C_DIS
LIN {X -0.186,Y -694.213,Z 840.436,A 0.000,B 0.000,C 90.000,E1 294.515} C_DIS
LIN {X 0.274,Y -694.472,Z 840.432,A 0.000,B 0.000,C 90.000,E1 293.770} C_DIS
LIN {X -0.144,Y -694.104,Z 840.430,A 0.000,B 0.000,C 90.000,E1 293.334} C_DIS
LIN {X 0.102,Y -693.705,Z 840.428,A 0.000,B 0.000,C 90.000,E1 293.078} C_DIS
LIN {X -0.320,Y -691.685,Z 840.426,A 0.000,B 0.000,C 90.000,E1 292.642} C_DIS
LIN {X -0.083,Y -690.273,Z 840.424,A 0.000,B 0.000,C 90.000,E1 292.386} C_DIS
LIN {X -0.229,Y -689.135,Z 840.424,A 0.000,B 0.000,C 90.000,E1 292.280} C_DIS
LIN {X -0.039,Y -683.220,Z 840.421,A 0.000,B 0.000,C 90.000,E1 291.844} C_DIS
LIN {X 0.300,Y -681.487,Z 840.421,A 0.000,B 0.000,C 90.000,E1 291.716} C_DIS
LIN {X -0.104,Y -679.091,Z 840.420,A 0.000,B 0.000,C 90.000,E1 291.663} C_DIS
LIN {X 0.045,Y -671.653,Z 840.419,A 0.000,B 0.000,C 90.000,E1 291.408} C_DIS
LIN {X -0.104,Y -665.025,Z 840.418,A 0.000,B 0.000,C 90.000,E1 291.280} C_DIS
LIN {X -0.280,Y -654.281,Z 840.417,A 0.000,B 0.000,C 90.000,E1 291.099} C_DIS
LIN {X 0.200,Y -648.090,Z 840.416,A 0.000,B 0.000,C 90.000,E1 290.918} C_DIS
LIN {X -0.189,Y -642.142,Z 840.415,A 0.000,B 0.000,C 90.000,E1 290.791} C_DIS
LIN {X -0.177,Y -635.326,Z 840.414,A 0.000,B 0.000,C 90.000,E1 290.536} C_DIS
LIN {X -0.303,Y -630.928,Z 840.413,A 0.000,B 0.000,C 90.000,E1 290.301} C_DIS
LIN {X 0.227,Y -630.848,Z 840.413,A 0.000,B 0.000,C 90.000,E1 290.248} C_DIS
LIN {X -0.221,Y -629.232,Z 840.411,A 0.000,B 0.000,C 90.000,E1 290.066} C_DIS
LIN {X -0.265,Y -629.212,Z 840.411,A 0.000,B 0.000,C 90.000,E1 290.066} C_DIS
LIN {X 0.093,Y -629.450,Z 840.410,A 0.000,B 0.000,C 90.000,E1 289.812} C_DIS
LIN {X -0.031,Y -632.111,Z 840.407,A 0.000,B 0.000,C 90.000,E1 289.214} C_DIS
LIN {X 0.209,Y -637.200,Z 840.402,A 0.000,B 0.000,C 90.000,E1 288.308} C_DIS
LIN {X 0.043,Y -639.201,Z 840.400,A 0.000,B 0.000,C 90.000,E1 287.946} C_DIS
LIN {X -0.266,Y -642.724,Z 840.396,A 0.000,B 0.000,C 90.000,E1 287.221} C_DIS
LIN {X 0.221,Y -644.899,Z 840.393,A 0.000,B 0.000,C 90.000,E1 286.677} C_DIS
LIN {X -0.080,Y -646.757,Z 840.390,A 0.000,B 0.000,C 90.000,E1 286.205} C_DIS
LIN {X 0.295,Y -649.288,Z 840.386,A 0.000,B 0.000,C 90.000,E1 285.426} C_DIS
LIN {X 0.027,Y -650.591,Z 840.383,A 0.000,B 0.000,C 90.000,E1 284.954} C_DIS
LIN {X -0.232,Y -651.816,Z 840.380,A 0.000,B 0.000,C 90.000,E1 284.481} C_DIS
LIN {X 0.028,Y -653.152,Z 840.376,A 0.000,B 0.000,C 90.000,E1 283.716} C_DIS
LIN {X -0.092,Y -653.576,Z 840.375,A 0.000,B 0.000,C 90.000,E1 283.480} C_DIS
LIN {X -0.331,Y -654.067,Z 840.372,A 0.000,B 0.000,C 90.000,E1 283.008} C_DIS
LIN {X -0.047,Y -654.393,Z 840.368,A 0.000,B 0.000,C 90.000,E1 282.243} C_DIS
LIN {X -0.284,Y -654.302,Z 840.365,A 0.000,B 0.000,C 90.000,E1 281.771} C_DIS
LIN {X -0.005,Y -653.820,Z 840.361,A 0.000,B 0.000,C 90.000,E1 281.007} C_DIS
LIN {X 0.269,Y -653.216,Z 840.358,A 0.000,B 0.000,C 90.000,E1 280.489} C_DIS
LIN {X 0.018,Y -652.348,Z 840.356,A 0.000,B 0.000,C 90.000,E1 280.018} C_DIS
LIN {X 0.290,Y -651.252,Z 840.353,A 0.000,B 0.000,C 90.000,E1 279.500} C_DIS
LIN {X 0.020,Y -649.723,Z 840.350,A 0.000,B 0.000,C 90.000,E1 279.029} C_DIS
LIN {X -0.220,Y -648.821,Z 840.349,A 0.000,B 0.000,C 90.000,E1 278.803} C_DIS
LIN {X 0.130,Y -646.700,Z 840.346,A 0.000,B 0.000,C 90.000,E1 278.276} C_DIS
LIN {X -0.268,Y -644.303,Z 840.343,A 0.000,B 0.000,C 90.000,E1 277.814} C_DIS
LIN {X -0.044,Y -641.489,Z 840.341,A 0.000,B 0.000,C 90.000,E1 277.296} C_DIS
LIN {X 0.030,Y -637.064,Z 840.337,A 0.000,B 0.000,C 90.000,E1 276.663} C_DIS
LIN {X 0.204,Y -633.069,Z 840.334,A 0.000,B 0.000,C 90.000,E1 276.144} C_DIS
LIN {X -0.199,Y -628.131,Z 840.332,A 0.000,B 0.000,C 90.000,E1 275.682} C_DIS
LIN {X 0.312,Y -625.355,Z 840.330,A 0.000,B 0.000,C 90.000,E1 275.391} C_DIS
LIN {X -0.269,Y -621.061,Z 840.328,A 0.000,B 0.000,C 90.000,E1 275.106} C_DIS
LIN {X -0.183,Y -617.784,Z 840.327,A 0.000,B 0.000,C 90.000,E1 274.878} C_DIS
LIN {X 0.044,Y -611.527,Z 840.325,A 0.000,B 0.000,C 90.000,E1 274.473} C_DIS
LIN {X -0.013,Y -604.563,Z 840.323,A 0.000,B 0.000,C 90.000,E1 274.131} C_DIS
LIN {X 0.281,Y -597.628,Z 840.321,A 0.000,B 0.000,C 90.000,E1 273.784} C_DIS
LIN {X 0.206,Y -588.822,Z 840.319,A 0.000,B 0.000,C 90.000,E1 273.440} C_DIS
LIN {X 0.040,Y -585.172,Z 840.319,A 0.000,B 0.000,C 90.000,E1 273.326} C_DIS
LIN {X 0.157,Y -579.088,Z 840.318,A 0.000,B 0.000,C 90.000,E1 273.154} C_DIS
LIN {X 0.096,Y -572.582,Z 840.317,A 0.000,B 0.000,C 90.000,E1 273.037} C_DIS
LIN {X -0.224,Y -570.301,Z 840.317,A 0.000,B 0.000,C 90.000,E1 273.037} C_DIS
LIN {X -0.150,Y -564.082,Z 840.317,A 0.000,B 0.000,C 90.000,E1 272.980} C_DIS
LIN {X 0.225,Y -556.726,Z 840.316,A 0.000,B 0.000,C 90.000,E1 272.922} C_DIS
LIN {X -0.111,Y -553.179,Z 840.316,A 0.000,B 0.000,C 90.000,E1 272.922} C_DIS
LIN {X 0.041,Y -550.545,Z 840.316,A 0.000,B 0.000,C 90.000,E1 272.808} C_DIS
LIN {X 0.003,Y -550.497,Z 840.316,A 0.000,B 0.000,C 90.000,E1 272.808} C_DIS
LIN {X -0.147,Y -549.517,Z 840.315,A 0.000,B 0.000,C 90.000,E1 272.636} C_DIS
LIN {X -0.115,Y -548.670,Z 840.313,A 0.000,B 0.000,C 90.000,E1 272.350} C_DIS
LIN {X 0.117,Y -547.704,Z 840.310,A 0.000,B 0.000,C 90.000,E1 271.776} C_DIS
LIN {X -0.160,Y -545.995,Z 840.301,A 0.000,B 0.000,C 90.000,E1 270.115} C_DIS
LIN {X 0.078,Y -544.747,Z 840.291,A 0.000,B 0.000,C 90.000,E1 268.396} C_DIS
LIN {X -0.279,Y -543.759,Z 840.283,A 0.000,B 0.000,C 90.000,E1 267.020} C_DIS
LIN {X -0.055,Y -542.595,Z 840.274,A 0.000,B 0.000,C 90.000,E1 265.298} C_DIS
LIN {X 0.180,Y -541.672,Z 840.266,A 0.000,B 0.000,C 90.000,E1 263.856} C_DIS
LIN {X -0.273,Y -540.973,Z 840.261,A 0.000,B 0.000,C 90.000,E1 263.053} C_DIS
LIN {X -0.005,Y -539.432,Z 840.252,A 0.000,B 0.000,C 90.000,E1 261.319} C_DIS
LIN {X -0.195,Y -538.106,Z 840.244,A 0.000,B 0.000,C 90.000,E1 259.916} C_DIS
LIN {X 0.092,Y -536.357,Z 840.234,A 0.000,B 0.000,C 90.000,E1 258.173} C_DIS
LIN {X 0.028,Y -534.604,Z 840.225,A 0.000,B 0.000,C 90.000,E1 256.464} C_DIS
LIN {X -0.160,Y -533.250,Z 840.219,A 0.000,B 0.000,C 90.000,E1 255.338} C_DIS
LIN {X 0.145,Y -531.941,Z 840.212,A 0.000,B 0.000,C 90.000,E1 254.157} C_DIS
LIN {X 0.272,Y -529.927,Z 840.203,A 0.000,B 0.000,C 90.000,E1 252.417} C_DIS
LIN {X 0.169,Y -528.119,Z 840.195,A 0.000,B 0.000,C 90.000,E1 250.986} C_DIS
LIN {X -0.122,Y -526.175,Z 840.186,A 0.000,B 0.000,C 90.000,E1 249.571} C_DIS
LIN {X 0.049,Y -524.170,Z 840.178,A 0.000,B 0.000,C 90.000,E1 248.103} C_DIS
LIN {X -0.105,Y -522.096,Z 840.170,A 0.000,B 0.000,C 90.000,E1 246.666} C_DIS
LIN {X 0.032,Y -520.349,Z 840.164,A 0.000,B 0.000,C 90.000,E1 245.485} C_DIS
LIN {X 0.022,Y -517.998,Z 840.156,A 0.000,B 0.000,C 90.000,E1 244.024} C_DIS
LIN {X 0.203,Y -515.442,Z 840.148,A 0.000,B 0.000,C 90.000,E1 242.538} C_DIS
LIN {X -0.114,Y -512.830,Z 840.139,A 0.000,B 0.000,C 90.000,E1 241.101} C_DIS
LIN {X -0.122,Y -510.716,Z 840.133,A 0.000,B 0.000,C 90.000,E1 239.921} C_DIS
LIN {X 0.059,Y -507.400,Z 840.123,A 0.000,B 0.000,C 90.000,E1 238.122} C_DIS
LIN {X 0.218,Y -505.029,Z 840.116,A 0.000,B 0.000,C 90.000,E1 236.914} C_DIS
LIN {X -0.087,Y -502.465,Z 840.110,A 0.000,B 0.000,C 90.000,E1 235.754} C_DIS
LIN {X -0.147,Y -499.745,Z 840.103,A 0.000,B 0.000,C 90.000,E1 234.562} C_DIS
LIN {X 0.040,Y -494.723,Z 840.091,A 0.000,B 0.000,C 90.000,E1 232.431} C_DIS
LIN {X -0.082,Y -492.644,Z 840.086,A 0.000,B 0.000,C 90.000,E1 231.537} C_DIS
LIN {X 0.155,Y -489.099,Z 840.078,A 0.000,B 0.000,C 90.000,E1 229.989} C_DIS
LIN {X -0.053,Y -485.627,Z 840.069,A 0.000,B 0.000,C 90.000,E1 228.485} C_DIS
LIN {X -0.173,Y -479.396,Z 840.054,A 0.000,B 0.000,C 90.000,E1 225.729} C_DIS
LIN {X -0.256,Y -476.080,Z 840.045,A 0.000,B 0.000,C 90.000,E1 224.190} C_DIS
LIN {X -0.197,Y -471.292,Z 840.033,A 0.000,B 0.000,C 90.000,E1 222.000} C_DIS
LIN {X 0.174,Y -468.657,Z 840.026,A 0.000,B 0.000,C 90.000,E1 220.701} C_DIS
LIN {X 0.013,Y -464.734,Z 840.016,A 0.000,B 0.000,C 90.000,E1 218.830} C_DIS
LIN {X -0.028,Y -462.079,Z 840.009,A 0.000,B 0.000,C 90.000,E1 217.569} C_DIS
LIN {X -0.027,Y -459.531,Z 840.002,A 0.000,B 0.000,C 90.000,E1 216.297} C_DIS
LIN {X 0.231,Y -454.023,Z 839.987,A 0.000,B 0.000,C 90.000,E1 213.706} C_DIS
LIN {X 0.110,Y -449.249,Z 839.975,A 0.000,B 0.000,C 90.000,E1 211.465} C_DIS
LIN {X 0.071,Y -443.852,Z 839.961,A 0.000,B 0.000,C 90.000,E1 208.871} C_DIS
LIN {X -0.134,Y -441.213,Z 839.953,A 0.000,B 0.000,C 90.000,E1 207.590} C_DIS
LIN {X 0.054,Y -437.972,Z 839.944,A 0.000,B 0.000,C 90.000,E1 205.924} C_DIS
LIN {X -0.007,Y -433.915,Z 839.933,A 0.000,B 0.000,C 90.000,E1 203.951} C_DIS
LIN {X 0.064,Y -428.640,Z 839.918,A 0.000,B 0.000,C 90.000,E1 201.280} C_DIS
LIN {X 0.081,Y -426.030,Z 839.911,A 0.000,B 0.000,C 90.000,E1 199.939} C_DIS
LIN {X 0.242,Y -422.757,Z 839.902,A 0.000,B 0.000,C 90.000,E1 198.236} C_DIS
LIN {X 0.013,Y -418.214,Z 839.888,A 0.000,B 0.000,C 90.000,E1 195.898} C_DIS
LIN {X 0.015,Y -415.578,Z 839.881,A 0.000,B 0.000,C 90.000,E1 194.537} C_DIS
LIN {X 0.046,Y -411.434,Z 839.869,A 0.000,B 0.000,C 90.000,E1 192.479} C_DIS
LIN {X -0.028,Y -407.486,Z 839.858,A 0.000,B 0.000,C 90.000,E1 190.423} C_DIS
LIN {X -0.016,Y -403.523,Z 839.846,A 0.000,B 0.000,C 90.000,E1 188.341} C_DIS
LIN {X -0.079,Y -400.111,Z 839.837,A 0.000,B 0.000,C 90.000,E1 186.606} C_DIS
LIN {X 0.006,Y -395.188,Z 839.821,A 0.000,B 0.000,C 90.000,E1 183.784} C_DIS
LIN {X 0.007,Y -391.920,Z 839.809,A 0.000,B 0.000,C 90.000,E1 181.661} C_DIS
LIN {X 0.121,Y -388.138,Z 839.793,A 0.000,B 0.000,C 90.000,E1 178.797} C_DIS
LIN {X -0.043,Y -385.324,Z 839.782,A 0.000,B 0.000,C 90.000,E1 176.674} C_DIS
LIN {X 0.140,Y -382.612,Z 839.770,A 0.000,B 0.000,C 90.000,E1 174.489} C_DIS
LIN {X 0.008,Y -378.726,Z 839.751,A 0.000,B 0.000,C 90.000,E1 171.254} C_DIS
LIN {X 0.050,Y -376.164,Z 839.737,A 0.000,B 0.000,C 90.000,E1 168.701} C_DIS
LIN {X -0.129,Y -374.074,Z 839.723,A 0.000,B 0.000,C 90.000,E1 166.172} C_DIS
LIN {X -0.143,Y -372.587,Z 839.711,A 0.000,B 0.000,C 90.000,E1 163.976} C_DIS
LIN {X -0.056,Y -372.001,Z 839.701,A 0.000,B 0.000,C 90.000,E1 162.127} C_DIS
LIN {X -0.100,Y -372.228,Z 839.690,A 0.000,B 0.000,C 90.000,E1 160.296} C_DIS
LIN {X -0.167,Y -372.573,Z 839.686,A 0.000,B 0.000,C 90.000,E1 159.571} C_DIS
LIN {X -0.131,Y -373.540,Z 839.680,A 0.000,B 0.000,C 90.000,E1 158.465} C_DIS
LIN {X -0.086,Y -374.910,Z 839.674,A 0.000,B 0.000,C 90.000,E1 157.358} C_DIS
LIN {X -0.013,Y -376.785,Z 839.669,A 0.000,B 0.000,C 90.000,E1 156.433} C_DIS
LIN {X -0.187,Y -378.127,Z 839.667,A 0.000,B 0.000,C 90.000,E1 156.049} C_DIS
LIN {X 0.082,Y -380.222,Z 839.663,A 0.000,B 0.000,C 90.000,E1 155.281} C_DIS
LIN {X 0.015,Y -385.215,Z 839.657,A 0.000,B 0.000,C 90.000,E1 154.332} C_DIS
LIN {X -0.041,Y -386.970,Z 839.656,A 0.000,B 0.000,C 90.000,E1 154.101} C_DIS
LIN {X 0.186,Y -391.065,Z 839.654,A 0.000,B 0.000,C 90.000,E1 153.640} C_DIS
LIN {X -0.023,Y -395.799,Z 839.652,A 0.000,B 0.000,C 90.000,E1 153.332} C_DIS
LIN {X -0.152,Y -399.529,Z 839.651,A 0.000,B 0.000,C 90.000,E1 153.127} C_DIS
LIN {X -0.052,Y -406.609,Z 839.649,A 0.000,B 0.000,C 90.000,E1 152.794} C_DIS
LIN {X 0.083,Y -414.101,Z 839.647,A 0.000,B 0.000,C 90.000,E1 152.487} C_DIS
LIN {X -0.153,Y -420.966,Z 839.646,A 0.000,B 0.000,C 90.000,E1 152.231} C_DIS
LIN {X -0.011,Y -427.120,Z 839.644,A 0.000,B 0.000,C 90.000,E1 151.897} C_DIS
LIN {X 0.097,Y -436.989,Z 839.641,A 0.000,B 0.000,C 90.000,E1 151.307} C_DIS
LIN {X 0.060,Y -443.521,Z 839.639,A 0.000,B 0.000,C 90.000,E1 150.923} C_DIS
LIN {X -0.095,Y -455.496,Z 839.633,A 0.000,B 0.000,C 90.000,E1 149.999} C_DIS
LIN {X 0.173,Y -461.345,Z 839.630,A 0.000,B 0.000,C 90.000,E1 149.459} C_DIS
LIN {X -0.007,Y -469.871,Z 839.626,A 0.000,B 0.000,C 90.000,E1 148.663} C_DIS
LIN {X -0.200,Y -472.588,Z 839.624,A 0.000,B 0.000,C 90.000,E1 148.408} C_DIS
LIN {X -0.011,Y -480.942,Z 839.620,A 0.000,B 0.000,C 90.000,E1 147.502} C_DIS
LIN {X 0.198,Y -489.726,Z 839.614,A 0.000,B 0.000,C 90.000,E1 146.421} C_DIS
LIN {X 0.283,Y -494.598,Z 839.610,A 0.000,B 0.000,C 90.000,E1 145.801} C_DIS
LIN {X -0.003,Y -498.906,Z 839.607,A 0.000,B 0.000,C 90.000,E1 145.229} C_DIS
LIN {X -0.075,Y -506.686,Z 839.600,A 0.000,B 0.000,C 90.000,E1 144.036} C_DIS
LIN {X -0.063,Y -511.349,Z 839.596,A 0.000,B 0.000,C 90.000,E1 143.290} C_DIS
LIN {X -0.124,Y -520.365,Z 839.588,A 0.000,B 0.000,C 90.000,E1 141.823} C_DIS
LIN {X -0.229,Y -523.834,Z 839.585,A 0.000,B 0.000,C 90.000,E1 141.251} C_DIS
LIN {X 0.143,Y -529.669,Z 839.579,A 0.000,B 0.000,C 90.000,E1 140.194} C_DIS
LIN {X -0.163,Y -536.631,Z 839.572,A 0.000,B 0.000,C 90.000,E1 138.933} C_DIS
LIN {X -0.198,Y -542.624,Z 839.565,A 0.000,B 0.000,C 90.000,E1 137.796} C_DIS
LIN {X 0.025,Y -549.243,Z 839.558,A 0.000,B 0.000,C 90.000,E1 136.500} C_DIS
LIN {X -0.094,Y -553.033,Z 839.555,A 0.000,B 0.000,C 90.000,E1 135.810} C_DIS
LIN {X -0.233,Y -555.218,Z 839.552,A 0.000,B 0.000,C 90.000,E1 135.405} C_DIS
LIN {X 0.207,Y -561.545,Z 839.545,A 0.000,B 0.000,C 90.000,E1 134.109} C_DIS
LIN {X 0.114,Y -563.537,Z 839.543,A 0.000,B 0.000,C 90.000,E1 133.704} C_DIS
LIN {X -0.144,Y -571.145,Z 839.534,A 0.000,B 0.000,C 90.000,E1 132.081} C_DIS
LIN {X 0.156,Y -576.645,Z 839.527,A 0.000,B 0.000,C 90.000,E1 130.825} C_DIS
LIN {X 0.168,Y -580.014,Z 839.522,A 0.000,B 0.000,C 90.000,E1 130.011} C_DIS
LIN {X 0.114,Y -585.245,Z 839.515,A 0.000,B 0.000,C 90.000,E1 128.669} C_DIS
LIN {X 0.048,Y -589.152,Z 839.509,A 0.000,B 0.000,C 90.000,E1 127.604} C_DIS
LIN {X 0.188,Y -591.594,Z 839.505,A 0.000,B 0.000,C 90.000,E1 126.790} C_DIS
LIN {X 0.211,Y -594.373,Z 839.499,A 0.000,B 0.000,C 90.000,E1 125.724} C_DIS
LIN {X 0.044,Y -596.137,Z 839.494,A 0.000,B 0.000,C 90.000,E1 124.945} C_DIS
LIN {X 0.385,Y -597.679,Z 839.490,A 0.000,B 0.000,C 90.000,E1 124.119} C_DIS
LIN {X 0.057,Y -599.730,Z 839.482,A 0.000,B 0.000,C 90.000,E1 122.832} C_DIS
LIN {X -0.153,Y -601.121,Z 839.477,A 0.000,B 0.000,C 90.000,E1 121.799} C_DIS
LIN {X -0.076,Y -601.923,Z 839.472,A 0.000,B 0.000,C 90.000,E1 121.003} C_DIS
LIN {X -0.055,Y -602.654,Z 839.466,A 0.000,B 0.000,C 90.000,E1 119.951} C_DIS
LIN {X -0.021,Y -602.909,Z 839.461,A 0.000,B 0.000,C 90.000,E1 118.899} C_DIS
LIN {X 0.076,Y -602.716,Z 839.456,A 0.000,B 0.000,C 90.000,E1 118.103} C_DIS
LIN {X -0.114,Y -602.288,Z 839.452,A 0.000,B 0.000,C 90.000,E1 117.334} C_DIS
LIN {X -0.036,Y -601.650,Z 839.447,A 0.000,B 0.000,C 90.000,E1 116.539} C_DIS
LIN {X 0.299,Y -600.866,Z 839.443,A 0.000,B 0.000,C 90.000,E1 115.720} C_DIS
LIN {X 0.159,Y -600.182,Z 839.440,A 0.000,B 0.000,C 90.000,E1 115.207} C_DIS
LIN {X 0.012,Y -599.207,Z 839.437,A 0.000,B 0.000,C 90.000,E1 114.695} C_DIS
LIN {X 0.079,Y -597.423,Z 839.433,A 0.000,B 0.000,C 90.000,E1 113.898} C_DIS
LIN {X 0.276,Y -593.679,Z 839.427,A 0.000,B 0.000,C 90.000,E1 112.823} C_DIS
LIN {X -0.098,Y -591.726,Z 839.425,A 0.000,B 0.000,C 90.000,E1 112.461} C_DIS
LIN {X -0.201,Y -590.289,Z 839.423,A 0.000,B 0.000,C 90.000,E1 112.206} C_DIS
LIN {X 0.291,Y -589.117,Z 839.423,A 0.000,B 0.000,C 90.000,E1 112.025} C_DIS
LIN {X 0.004,Y -584.947,Z 839.420,A 0.000,B 0.000,C 90.000,E1 111.663} C_DIS
LIN {X 0.047,Y -583.281,Z 839.420,A 0.000,B 0.000,C 90.000,E1 111.535} C_DIS
LIN {X 0.290,Y -576.833,Z 839.417,A 0.000,B 0.000,C 90.000,E1 111.099} C_DIS
LIN {X 0.047,Y -571.586,Z 839.416,A 0.000,B 0.000,C 90.000,E1 110.844} C_DIS
LIN {X -0.277,Y -566.059,Z 839.413,A 0.000,B 0.000,C 90.000,E1 110.429} C_DIS
LIN {X 0.239,Y -565.027,Z 839.413,A 0.000,B 0.000,C 90.000,E1 110.248} C_DIS
LIN {X -0.094,Y -563.450,Z 839.409,A 0.000,B 0.000,C 90.000,E1 109.631} C_DIS
LIN {X -0.170,Y -562.610,Z 839.406,A 0.000,B 0.000,C 90.000,E1 109.087} C_DIS
LIN {X -0.269,Y -561.697,Z 839.400,A 0.000,B 0.000,C 90.000,E1 108.000} C_DIS
LIN {X -0.321,Y -562.846,Z 839.369,A 0.000,B 0.000,C 90.000,E1 102.479} C_DIS
LIN {X -0.295,Y -564.079,Z 839.358,A 0.000,B 0.000,C 90.000,E1 100.546} C_DIS
LIN {X -0.125,Y -565.093,Z 839.351,A 0.000,B 0.000,C 90.000,E1 99.151} C_DIS
LIN {X 0.060,Y -566.005,Z 839.343,A 0.000,B 0.000,C 90.000,E1 97.757} C_DIS
LIN {X 0.178,Y -566.884,Z 839.336,A 0.000,B 0.000,C 90.000,E1 96.372} C_DIS
LIN {X 0.254,Y -567.605,Z 839.328,A 0.000,B 0.000,C 90.000,E1 94.992} C_DIS
LIN {X -0.105,Y -568.242,Z 839.319,A 0.000,B 0.000,C 90.000,E1 93.383} C_DIS
LIN {X -0.036,Y -568.678,Z 839.311,A 0.000,B 0.000,C 90.000,E1 92.007} C_DIS
LIN {X 0.162,Y -569.181,Z 839.302,A 0.000,B 0.000,C 90.000,E1 90.344} C_DIS
LIN {X -0.212,Y -569.587,Z 839.293,A 0.000,B 0.000,C 90.000,E1 88.740} C_DIS
LIN {X 0.155,Y -569.983,Z 839.282,A 0.000,B 0.000,C 90.000,E1 86.788} C_DIS
LIN {X -0.033,Y -570.310,Z 839.272,A 0.000,B 0.000,C 90.000,E1 84.894} C_DIS
LIN {X 0.099,Y -570.575,Z 839.264,A 0.000,B 0.000,C 90.000,E1 83.514} C_DIS
LIN {X 0.100,Y -571.042,Z 839.253,A 0.000,B 0.000,C 90.000,E1 81.602} C_DIS
LIN {X 0.117,Y -571.575,Z 839.243,A 0.000,B 0.000,C 90.000,E1 79.690} C_DIS
LIN {X -0.038,Y -572.086,Z 839.235,A 0.000,B 0.000,C 90.000,E1 78.342} C_DIS
LIN {X -0.178,Y -572.464,Z 839.228,A 0.000,B 0.000,C 90.000,E1 76.992} C_DIS
LIN {X 0.018,Y -572.860,Z 839.219,A 0.000,B 0.000,C 90.000,E1 75.338} C_DIS
LIN {X 0.040,Y -572.996,Z 839.214,A 0.000,B 0.000,C 90.000,E1 74.519} C_DIS
LIN {X -0.168,Y -573.121,Z 839.205,A 0.000,B 0.000,C 90.000,E1 72.906} C_DIS
LIN {X -0.199,Y -573.084,Z 839.196,A 0.000,B 0.000,C 90.000,E1 71.275} C_DIS
LIN {X -0.037,Y -572.933,Z 839.187,A 0.000,B 0.000,C 90.000,E1 69.625} C_DIS
LIN {X 0.311,Y -572.875,Z 839.182,A 0.000,B 0.000,C 90.000,E1 68.773} C_DIS
LIN {X 0.314,Y -572.660,Z 839.175,A 0.000,B 0.000,C 90.000,E1 67.411} C_DIS
LIN {X -0.214,Y -572.337,Z 839.167,A 0.000,B 0.000,C 90.000,E1 66.102} C_DIS
LIN {X 0.007,Y -571.837,Z 839.160,A 0.000,B 0.000,C 90.000,E1 64.717} C_DIS
LIN {X 0.040,Y -571.139,Z 839.151,A 0.000,B 0.000,C 90.000,E1 63.076} C_DIS
LIN {X -0.033,Y -570.556,Z 839.143,A 0.000,B 0.000,C 90.000,E1 61.719} C_DIS
LIN {X -0.272,Y -570.120,Z 839.138,A 0.000,B 0.000,C 90.000,E1 60.923} C_DIS
LIN {X 0.092,Y -569.236,Z 839.132,A 0.000,B 0.000,C 90.000,E1 59.793} C_DIS
LIN {X -0.337,Y -568.144,Z 839.126,A 0.000,B 0.000,C 90.000,E1 58.742} C_DIS
LIN {X 0.293,Y -566.868,Z 839.120,A 0.000,B 0.000,C 90.000,E1 57.582} C_DIS
LIN {X 0.123,Y -565.456,Z 839.114,A 0.000,B 0.000,C 90.000,E1 56.501} C_DIS
LIN {X 0.134,Y -564.224,Z 839.109,A 0.000,B 0.000,C 90.000,E1 55.674} C_DIS
LIN {X -0.226,Y -562.316,Z 839.103,A 0.000,B 0.000,C 90.000,E1 54.609} C_DIS
LIN {X -0.250,Y -560.729,Z 839.099,A 0.000,B 0.000,C 90.000,E1 53.783} C_DIS
LIN {X 0.125,Y -558.278,Z 839.093,A 0.000,B 0.000,C 90.000,E1 52.637} C_DIS
LIN {X -0.141,Y -556.946,Z 839.089,A 0.000,B 0.000,C 90.000,E1 52.110} C_DIS
LIN {X 0.101,Y -554.681,Z 839.085,A 0.000,B 0.000,C 90.000,E1 51.251} C_DIS
LIN {X -0.184,Y -553.053,Z 839.082,A 0.000,B 0.000,C 90.000,E1 50.723} C_DIS
LIN {X 0.006,Y -550.335,Z 839.077,A 0.000,B 0.000,C 90.000,E1 49.865} C_DIS
LIN {X 0.096,Y -547.234,Z 839.072,A 0.000,B 0.000,C 90.000,E1 49.013} C_DIS
LIN {X -0.236,Y -544.996,Z 839.069,A 0.000,B 0.000,C 90.000,E1 48.485} C_DIS
LIN {X -0.025,Y -541.945,Z 839.065,A 0.000,B 0.000,C 90.000,E1 47.757} C_DIS
LIN {X -0.206,Y -538.528,Z 839.061,A 0.000,B 0.000,C 90.000,E1 47.067} C_DIS
LIN {X 0.157,Y -535.631,Z 839.058,A 0.000,B 0.000,C 90.000,E1 46.458} C_DIS
LIN {X 0.108,Y -532.429,Z 839.055,A 0.000,B 0.000,C 90.000,E1 45.891} C_DIS
LIN {X 0.203,Y -527.818,Z 839.051,A 0.000,B 0.000,C 90.000,E1 45.162} C_DIS
LIN {X 0.101,Y -523.916,Z 839.048,A 0.000,B 0.000,C 90.000,E1 44.595} C_DIS
LIN {X -0.029,Y -519.601,Z 839.045,A 0.000,B 0.000,C 90.000,E1 44.028} C_DIS
LIN {X -0.052,Y -513.784,Z 839.041,A 0.000,B 0.000,C 90.000,E1 43.299} C_DIS
LIN {X 0.117,Y -508.797,Z 839.037,A 0.000,B 0.000,C 90.000,E1 42.690} C_DIS
LIN {X -0.197,Y -502.143,Z 839.033,A 0.000,B 0.000,C 90.000,E1 42.000} C_DIS
LIN {X 0.153,Y -496.580,Z 839.030,A 0.000,B 0.000,C 90.000,E1 41.391} C_DIS
LIN {X -0.038,Y -490.806,Z 839.027,A 0.000,B 0.000,C 90.000,E1 40.862} C_DIS
LIN {X -0.003,Y -486.305,Z 839.025,A 0.000,B 0.000,C 90.000,E1 40.458} C_DIS
LIN {X -0.062,Y -479.010,Z 839.021,A 0.000,B 0.000,C 90.000,E1 39.850} C_DIS
LIN {X -0.151,Y -469.695,Z 839.017,A 0.000,B 0.000,C 90.000,E1 39.116} C_DIS
LIN {X -0.174,Y -458.920,Z 839.013,A 0.000,B 0.000,C 90.000,E1 38.302} C_DIS
LIN {X -0.042,Y -449.425,Z 839.009,A 0.000,B 0.000,C 90.000,E1 37.569} C_DIS
LIN {X 0.115,Y -438.267,Z 839.004,A 0.000,B 0.000,C 90.000,E1 36.710} C_DIS
LIN {X -0.171,Y -416.878,Z 838.995,A 0.000,B 0.000,C 90.000,E1 35.025} C_DIS
LIN {X -0.164,Y -403.338,Z 838.988,A 0.000,B 0.000,C 90.000,E1 33.785} C_DIS
LIN {X -0.012,Y -399.672,Z 838.985,A 0.000,B 0.000,C 90.000,E1 33.372} C_DIS
LIN {X 0.008,Y -397.123,Z 838.984,A 0.000,B 0.000,C 90.000,E1 33.038} C_DIS
LIN {X 0.018,Y -395.042,Z 838.982,A 0.000,B 0.000,C 90.000,E1 32.704} C_DIS
LIN {X -0.005,Y -395.027,Z 838.982,A 0.000,B 0.000,C 90.000,E1 32.704} C_DIS
LIN {X -0.034,Y -393.957,Z 838.978,A 0.000,B 0.000,C 90.000,E1 31.957} C_DIS
LIN {X 0.100,Y -391.952,Z 838.972,A 0.000,B 0.000,C 90.000,E1 30.875} C_DIS
LIN {X 0.155,Y -390.959,Z 838.969,A 0.000,B 0.000,C 90.000,E1 30.335} C_DIS
LIN {X 0.096,Y -391.422,Z 838.960,A 0.000,B 0.000,C 90.000,E1 28.743} C_DIS
LIN {X -0.139,Y -392.453,Z 838.950,A 0.000,B 0.000,C 90.000,E1 27.001} C_DIS
LIN {X 0.091,Y -394.413,Z 838.934,A 0.000,B 0.000,C 90.000,E1 24.131} C_DIS
LIN {X -0.009,Y -396.117,Z 838.922,A 0.000,B 0.000,C 90.000,E1 22.025} C_DIS
LIN {X -0.061,Y -398.643,Z 838.907,A 0.000,B 0.000,C 90.000,E1 19.214} C_DIS
LIN {X 0.126,Y -401.354,Z 838.893,A 0.000,B 0.000,C 90.000,E1 16.732} C_DIS
LIN {X 0.134,Y -406.024,Z 838.874,A 0.000,B 0.000,C 90.000,E1 13.244} C_DIS
LIN {X 0.053,Y -410.937,Z 838.856,A 0.000,B 0.000,C 90.000,E1 10.141} C_DIS
LIN {X -0.183,Y -413.866,Z 838.847,A 0.000,B 0.000,C 90.000,E1 8.454} C_DIS
LIN {X 0.035,Y -417.517,Z 838.835,A 0.000,B 0.000,C 90.000,E1 6.372} C_DIS
LIN {X -0.076,Y -422.527,Z 838.820,A 0.000,B 0.000,C 90.000,E1 3.669} C_DIS
LIN {X 0.054,Y -429.523,Z 838.802,A 0.000,B 0.000,C 90.000,E1 0.286} C_DIS
LIN {X 0.146,Y -434.531,Z 838.790,A 0.000,B 0.000,C 90.000,E1 358.108} C_DIS
LIN {X -0.130,Y -439.323,Z 838.779,A 0.000,B 0.000,C 90.000,E1 356.159} C_DIS
LIN {X 0.036,Y -446.035,Z 838.764,A 0.000,B 0.000,C 90.000,E1 353.514} C_DIS
LIN {X -0.059,Y -447.819,Z 838.760,A 0.000,B 0.000,C 90.000,E1 352.875} C_DIS
LIN {X -0.064,Y -450.641,Z 838.756,A 0.000,B 0.000,C 90.000,E1 352.064} C_DIS
LIN {X 0.198,Y -452.697,Z 838.754,A 0.000,B 0.000,C 90.000,E1 351.602} C_DIS
LIN {X -0.182,Y -453.599,Z 838.753,A 0.000,B 0.000,C 90.000,E1 351.489} C_DIS
LIN {X -0.115,Y -454.818,Z 838.752,A 0.000,B 0.000,C 90.000,E1 351.319} C_DIS
LIN {X -0.117,Y -457.672,Z 838.750,A 0.000,B 0.000,C 90.000,E1 351.027} C_DIS
LIN {X 0.115,Y -460.861,Z 838.749,A 0.000,B 0.000,C 90.000,E1 350.735} C_DIS
LIN {X 0.104,Y -466.041,Z 838.747,A 0.000,B 0.000,C 90.000,E1 350.387} C_DIS
LIN {X 0.166,Y -481.303,Z 838.742,A 0.000,B 0.000,C 90.000,E1 349.511} C_DIS
LIN {X 0.024,Y -489.442,Z 838.739,A 0.000,B 0.000,C 90.000,E1 349.050} C_DIS
LIN {X 0.006,Y -500.618,Z 838.735,A 0.000,B 0.000,C 90.000,E1 348.342} C_DIS
LIN {X 0.138,Y -510.063,Z 838.732,A 0.000,B 0.000,C 90.000,E1 347.701} C_DIS
LIN {X 0.119,Y -517.792,Z 838.729,A 0.000,B 0.000,C 90.000,E1 347.173} C_DIS
LIN {X 0.082,Y -528.603,Z 838.725,A 0.000,B 0.000,C 90.000,E1 346.408} C_DIS
LIN {X -0.107,Y -537.500,Z 838.721,A 0.000,B 0.000,C 90.000,E1 345.755} C_DIS
LIN {X -0.055,Y -546.085,Z 838.717,A 0.000,B 0.000,C 90.000,E1 345.046} C_DIS
LIN {X -0.160,Y -553.055,Z 838.714,A 0.000,B 0.000,C 90.000,E1 344.448} C_DIS
LIN {X 0.312,Y -559.673,Z 838.710,A 0.000,B 0.000,C 90.000,E1 343.795} C_DIS
LIN {X -0.234,Y -566.032,Z 838.707,A 0.000,B 0.000,C 90.000,E1 343.196} C_DIS
LIN {X -0.203,Y -571.021,Z 838.704,A 0.000,B 0.000,C 90.000,E1 342.653} C_DIS
LIN {X 0.052,Y -576.992,Z 838.700,A 0.000,B 0.000,C 90.000,E1 341.945} C_DIS
LIN {X 0.151,Y -580.328,Z 838.698,A 0.000,B 0.000,C 90.000,E1 341.529} C_DIS
LIN {X -0.362,Y -584.481,Z 838.695,A 0.000,B 0.000,C 90.000,E1 341.040} C_DIS
LIN {X 0.061,Y -591.421,Z 838.689,A 0.000,B 0.000,C 90.000,E1 340.061} C_DIS
LIN {X 0.021,Y -597.401,Z 838.684,A 0.000,B 0.000,C 90.000,E1 339.135} C_DIS
LIN {X -0.205,Y -603.821,Z 838.678,A 0.000,B 0.000,C 90.000,E1 338.103} C_DIS
LIN {X -0.176,Y -611.265,Z 838.671,A 0.000,B 0.000,C 90.000,E1 336.794} C_DIS
LIN {X 0.294,Y -614.851,Z 838.667,A 0.000,B 0.000,C 90.000,E1 336.102} C_DIS
LIN {X -0.040,Y -620.250,Z 838.662,A 0.000,B 0.000,C 90.000,E1 335.101} C_DIS
LIN {X -0.046,Y -624.708,Z 838.657,A 0.000,B 0.000,C 90.000,E1 334.204} C_DIS
LIN {X 0.015,Y -629.523,Z 838.651,A 0.000,B 0.000,C 90.000,E1 333.179} C_DIS
LIN {X 0.132,Y -634.010,Z 838.645,A 0.000,B 0.000,C 90.000,E1 332.153} C_DIS
LIN {X -0.257,Y -638.227,Z 838.640,A 0.000,B 0.000,C 90.000,E1 331.179} C_DIS
LIN {X 0.276,Y -642.290,Z 838.634,A 0.000,B 0.000,C 90.000,E1 330.127} C_DIS
LIN {X -0.019,Y -646.099,Z 838.629,A 0.000,B 0.000,C 90.000,E1 329.154} C_DIS
LIN {X 0.056,Y -649.585,Z 838.623,A 0.000,B 0.000,C 90.000,E1 328.152} C_DIS
LIN {X 0.063,Y -653.700,Z 838.616,A 0.000,B 0.000,C 90.000,E1 326.914} C_DIS
LIN {X 0.141,Y -655.950,Z 838.612,A 0.000,B 0.000,C 90.000,E1 326.167} C_DIS
LIN {X 0.160,Y -658.727,Z 838.607,A 0.000,B 0.000,C 90.000,E1 325.182} C_DIS
LIN {X -0.259,Y -660.705,Z 838.603,A 0.000,B 0.000,C 90.000,E1 324.482} C_DIS
LIN {X -0.176,Y -663.115,Z 838.597,A 0.000,B 0.000,C 90.000,E1 323.497} C_DIS
LIN {X 0.336,Y -665.205,Z 838.592,A 0.000,B 0.000,C 90.000,E1 322.477} C_DIS
LIN {X -0.053,Y -667.129,Z 838.586,A 0.000,B 0.000,C 90.000,E1 321.537} C_DIS
LIN {X -0.001,Y -668.846,Z 838.581,A 0.000,B 0.000,C 90.000,E1 320.561} C_DIS
LIN {X 0.159,Y -671.068,Z 838.573,A 0.000,B 0.000,C 90.000,E1 319.094} C_DIS
LIN {X 0.303,Y -673.608,Z 838.563,A 0.000,B 0.000,C 90.000,E1 317.391} C_DIS
LIN {X -0.091,Y -674.604,Z 838.559,A 0.000,B 0.000,C 90.000,E1 316.701} C_DIS
LIN {X 0.107,Y -676.729,Z 838.550,A 0.000,B 0.000,C 90.000,E1 315.000} C_DIS
LIN {X 0.282,Y -678.018,Z 838.543,A 0.000,B 0.000,C 90.000,E1 313.785} C_DIS
LIN {X 0.005,Y -679.313,Z 838.537,A 0.000,B 0.000,C 90.000,E1 312.609} C_DIS
LIN {X 0.295,Y -680.829,Z 838.529,A 0.000,B 0.000,C 90.000,E1 311.148} C_DIS
LIN {X 0.167,Y -682.219,Z 838.521,A 0.000,B 0.000,C 90.000,E1 309.725} C_DIS
LIN {X -0.328,Y -683.708,Z 838.512,A 0.000,B 0.000,C 90.000,E1 308.096} C_DIS
LIN {X -0.292,Y -684.936,Z 838.504,A 0.000,B 0.000,C 90.000,E1 306.664} C_DIS
LIN {X -0.235,Y -686.088,Z 838.496,A 0.000,B 0.000,C 90.000,E1 305.231} C_DIS
LIN {X 0.006,Y -687.073,Z 838.488,A 0.000,B 0.000,C 90.000,E1 303.785} C_DIS
LIN {X -0.100,Y -688.224,Z 838.479,A 0.000,B 0.000,C 90.000,E1 302.133} C_DIS
LIN {X -0.192,Y -689.287,Z 838.471,A 0.000,B 0.000,C 90.000,E1 300.718} C_DIS
LIN {X 0.088,Y -690.922,Z 838.459,A 0.000,B 0.000,C 90.000,E1 298.565} C_DIS
LIN {X 0.305,Y -692.075,Z 838.451,A 0.000,B 0.000,C 90.000,E1 297.129} C_DIS
LIN {X -0.157,Y -693.540,Z 838.442,A 0.000,B 0.000,C 90.000,E1 295.515} C_DIS
LIN {X -0.135,Y -694.512,Z 838.435,A 0.000,B 0.000,C 90.000,E1 294.335} C_DIS
LIN {X 0.363,Y -694.636,Z 838.433,A 0.000,B 0.000,C 90.000,E1 293.823} C_DIS
LIN {X -0.304,Y -694.533,Z 838.431,A 0.000,B 0.000,C 90.000,E1 293.643} C_DIS
LIN {X 0.189,Y -693.921,Z 838.429,A 0.000,B 0.000,C 90.000,E1 293.131} C_DIS
LIN {X 0.162,Y -693.056,Z 838.427,A 0.000,B 0.000,C 90.000,E1 292.898} C_DIS
LIN {X -0.381,Y -691.234,Z 838.425,A 0.000,B 0.000,C 90.000,E1 292.589} C_DIS
LIN {X -0.261,Y -690.560,Z 838.425,A 0.000,B 0.000,C 90.000,E1 292.461} C_DIS
LIN {X -0.145,Y -689.616,Z 838.424,A 0.000,B 0.000,C 90.000,E1 292.333} C_DIS
LIN {X -0.029,Y -688.210,Z 838.423,A 0.000,B 0.000,C 90.000,E1 292.206} C_DIS
LIN {X 0.224,Y -682.128,Z 838.421,A 0.000,B 0.000,C 90.000,E1 291.770} C_DIS
LIN {X -0.272,Y -679.915,Z 838.421,A 0.000,B 0.000,C 90.000,E1 291.716} C_DIS
LIN {X -0.182,Y -669.987,Z 838.419,A 0.000,B 0.000,C 90.000,E1 291.408} C_DIS
LIN {X -0.286,Y -663.226,Z 838.418,A 0.000,B 0.000,C 90.000,E1 291.280} C_DIS
LIN {X 0.045,Y -654.325,Z 838.417,A 0.000,B 0.000,C 90.000,E1 291.099} C_DIS
LIN {X 0.006,Y -648.239,Z 838.417,A 0.000,B 0.000,C 90.000,E1 290.972} C_DIS
LIN {X 0.288,Y -642.239,Z 838.416,A 0.000,B 0.000,C 90.000,E1 290.791} C_DIS
LIN {X 0.253,Y -633.489,Z 838.414,A 0.000,B 0.000,C 90.000,E1 290.482} C_DIS
LIN {X -0.075,Y -629.571,Z 838.413,A 0.000,B 0.000,C 90.000,E1 290.301} C_DIS
LIN {X 0.115,Y -627.373,Z 838.412,A 0.000,B 0.000,C 90.000,E1 290.066} C_DIS
LIN {X 0.072,Y -627.336,Z 838.412,A 0.000,B 0.000,C 90.000,E1 290.066} C_DIS
LIN {X -0.056,Y -627.215,Z 838.411,A 0.000,B 0.000,C 90.000,E1 289.939} C_DIS
LIN {X -0.163,Y -627.764,Z 838.410,A 0.000,B 0.000,C 90.000,E1 289.758} C_DIS
LIN {X -0.375,Y -629.338,Z 838.408,A 0.000,B 0.000,C 90.000,E1 289.396} C_DIS
LIN {X 0.221,Y -631.392,Z 838.406,A 0.000,B 0.000,C 90.000,E1 288.960} C_DIS
LIN {X 0.282,Y -633.545,Z 838.404,A 0.000,B 0.000,C 90.000,E1 288.598} C_DIS
LIN {X -0.090,Y -637.096,Z 838.400,A 0.000,B 0.000,C 90.000,E1 288.000} C_DIS
LIN {X 0.189,Y -640.671,Z 838.396,A 0.000,B 0.000,C 90.000,E1 287.221} C_DIS
LIN {X -0.112,Y -643.786,Z 838.392,A 0.000,B 0.000,C 90.000,E1 286.496} C_DIS
LIN {X 0.083,Y -647.291,Z 838.386,A 0.000,B 0.000,C 90.000,E1 285.481} C_DIS
LIN {X -0.061,Y -648.030,Z 838.385,A 0.000,B 0.000,C 90.000,E1 285.245} C_DIS
LIN {X 0.022,Y -650.357,Z 838.379,A 0.000,B 0.000,C 90.000,E1 284.245} C_DIS
LIN {X -0.109,Y -650.831,Z 838.378,A 0.000,B 0.000,C 90.000,E1 284.008} C_DIS
LIN {X -0.365,Y -651.583,Z 838.375,A 0.000,B 0.000,C 90.000,E1 283.536} C_DIS
LIN {X -0.106,Y -652.223,Z 838.371,A 0.000,B 0.000,C 90.000,E1 282.771} C_DIS
LIN {X 0.282,Y -652.436,Z 838.368,A 0.000,B 0.000,C 90.000,E1 282.243} C_DIS
LIN {X 0.033,Y -652.312,Z 838.365,A 0.000,B 0.000,C 90.000,E1 281.771} C_DIS
LIN {X 0.292,Y -651.784,Z 838.361,A 0.000,B 0.000,C 90.000,E1 281.007} C_DIS
LIN {X -0.089,Y -651.138,Z 838.359,A 0.000,B 0.000,C 90.000,E1 280.546} C_DIS
LIN {X 0.286,Y -650.227,Z 838.356,A 0.000,B 0.000,C 90.000,E1 280.018} C_DIS
LIN {X -0.097,Y -649.091,Z 838.353,A 0.000,B 0.000,C 90.000,E1 279.557} C_DIS
LIN {X 0.259,Y -647.516,Z 838.350,A 0.000,B 0.000,C 90.000,E1 279.029} C_DIS
LIN {X -0.137,Y -645.600,Z 838.348,A 0.000,B 0.000,C 90.000,E1 278.568} C_DIS
LIN {X -0.029,Y -642.745,Z 838.344,A 0.000,B 0.000,C 90.000,E1 277.936} C_DIS
LIN {X -0.320,Y -640.519,Z 838.342,A 0.000,B 0.000,C 90.000,E1 277.587} C_DIS
LIN {X 0.011,Y -638.129,Z 838.340,A 0.000,B 0.000,C 90.000,E1 277.182} C_DIS
LIN {X 0.192,Y -634.633,Z 838.337,A 0.000,B 0.000,C 90.000,E1 276.663} C_DIS
LIN {X -0.278,Y -630.297,Z 838.334,A 0.000,B 0.000,C 90.000,E1 276.201} C_DIS
LIN {X 0.058,Y -626.630,Z 838.332,A 0.000,B 0.000,C 90.000,E1 275.796} C_DIS
LIN {X -0.200,Y -623.692,Z 838.331,A 0.000,B 0.000,C 90.000,E1 275.568} C_DIS
LIN {X -0.005,Y -617.982,Z 838.328,A 0.000,B 0.000,C 90.000,E1 275.106} C_DIS
LIN {X 0.047,Y -611.388,Z 838.326,A 0.000,B 0.000,C 90.000,E1 274.702} C_DIS
LIN {X 0.207,Y -606.304,Z 838.325,A 0.000,B 0.000,C 90.000,E1 274.416} C_DIS
LIN {X 0.251,Y -597.746,Z 838.322,A 0.000,B 0.000,C 90.000,E1 274.012} C_DIS
LIN {X 0.205,Y -590.538,Z 838.321,A 0.000,B 0.000,C 90.000,E1 273.726} C_DIS
LIN {X -0.061,Y -585.382,Z 838.320,A 0.000,B 0.000,C 90.000,E1 273.555} C_DIS
LIN {X -0.034,Y -579.238,Z 838.319,A 0.000,B 0.000,C 90.000,E1 273.383} C_DIS
LIN {X -0.142,Y -572.720,Z 838.318,A 0.000,B 0.000,C 90.000,E1 273.269} C_DIS
LIN {X -0.152,Y -567.264,Z 838.318,A 0.000,B 0.000,C 90.000,E1 273.212} C_DIS
LIN {X 0.159,Y -562.842,Z 838.318,A 0.000,B 0.000,C 90.000,E1 273.154} C_DIS
LIN {X -0.111,Y -556.135,Z 838.318,A 0.000,B 0.000,C 90.000,E1 273.154} C_DIS
LIN {X -0.242,Y -553.443,Z 838.317,A 0.000,B 0.000,C 90.000,E1 273.151} C_DIS
LIN {X -0.140,Y -550.609,Z 838.317,A 0.000,B 0.000,C 90.000,E1 273.037} C_DIS
LIN {X -0.177,Y -550.561,Z 838.317,A 0.000,B 0.000,C 90.000,E1 273.037} C_DIS
LIN {X -0.218,Y -549.654,Z 838.316,A 0.000,B 0.000,C 90.000,E1 272.865} C_DIS
LIN {X 0.132,Y -548.738,Z 838.314,A 0.000,B 0.000,C 90.000,E1 272.522} C_DIS
LIN {X -0.215,Y -547.834,Z 838.311,A 0.000,B 0.000,C 90.000,E1 272.007} C_DIS
LIN {X -0.228,Y -544.921,Z 838.292,A 0.000,B 0.000,C 90.000,E1 268.625} C_DIS
LIN {X -0.006,Y -543.730,Z 838.283,A 0.000,B 0.000,C 90.000,E1 266.906} C_DIS
LIN {X 0.215,Y -542.578,Z 838.273,A 0.000,B 0.000,C 90.000,E1 265.184} C_DIS
LIN {X -0.162,Y -541.855,Z 838.267,A 0.000,B 0.000,C 90.000,E1 264.090} C_DIS
LIN {X -0.013,Y -541.203,Z 838.262,A 0.000,B 0.000,C 90.000,E1 263.223} C_DIS
LIN {X -0.199,Y -539.386,Z 838.251,A 0.000,B 0.000,C 90.000,E1 261.254} C_DIS
LIN {X 0.058,Y -538.046,Z 838.243,A 0.000,B 0.000,C 90.000,E1 259.803} C_DIS
LIN {X -0.078,Y -536.308,Z 838.234,A 0.000,B 0.000,C 90.000,E1 258.105} C_DIS
LIN {X -0.256,Y -534.548,Z 838.224,A 0.000,B 0.000,C 90.000,E1 256.408} C_DIS
LIN {X 0.070,Y -533.205,Z 838.218,A 0.000,B 0.000,C 90.000,E1 255.227} C_DIS
LIN {X 0.038,Y -531.566,Z 838.210,A 0.000,B 0.000,C 90.000,E1 253.795} C_DIS
LIN {X -0.021,Y -529.888,Z 838.202,A 0.000,B 0.000,C 90.000,E1 252.362} C_DIS
LIN {X 0.044,Y -528.096,Z 838.194,A 0.000,B 0.000,C 90.000,E1 250.913} C_DIS
LIN {X 0.253,Y -526.114,Z 838.186,A 0.000,B 0.000,C 90.000,E1 249.444} C_DIS
LIN {X 0.259,Y -524.508,Z 838.180,A 0.000,B 0.000,C 90.000,E1 248.284} C_DIS
LIN {X -0.094,Y -522.470,Z 838.172,A 0.000,B 0.000,C 90.000,E1 246.869} C_DIS
LIN {X 0.256,Y -520.726,Z 838.165,A 0.000,B 0.000,C 90.000,E1 245.665} C_DIS
LIN {X 0.032,Y -518.394,Z 838.157,A 0.000,B 0.000,C 90.000,E1 244.229} C_DIS
LIN {X 0.089,Y -516.391,Z 838.150,A 0.000,B 0.000,C 90.000,E1 243.050} C_DIS
LIN {X 0.000,Y -512.730,Z 838.139,A 0.000,B 0.000,C 90.000,E1 241.001} C_DIS
LIN {X -0.121,Y -510.046,Z 838.131,A 0.000,B 0.000,C 90.000,E1 239.537} C_DIS
LIN {X 0.034,Y -506.687,Z 838.121,A 0.000,B 0.000,C 90.000,E1 237.740} C_DIS
LIN {X 0.140,Y -504.878,Z 838.116,A 0.000,B 0.000,C 90.000,E1 236.834} C_DIS
LIN {X -0.164,Y -502.311,Z 838.109,A 0.000,B 0.000,C 90.000,E1 235.674} C_DIS
LIN {X -0.223,Y -499.575,Z 838.103,A 0.000,B 0.000,C 90.000,E1 234.482} C_DIS
LIN {X 0.102,Y -495.299,Z 838.093,A 0.000,B 0.000,C 90.000,E1 232.637} C_DIS
LIN {X -0.157,Y -492.475,Z 838.086,A 0.000,B 0.000,C 90.000,E1 231.457} C_DIS
LIN {X -0.076,Y -489.613,Z 838.079,A 0.000,B 0.000,C 90.000,E1 230.231} C_DIS
LIN {X -0.104,Y -486.860,Z 838.072,A 0.000,B 0.000,C 90.000,E1 229.013} C_DIS
LIN {X -0.172,Y -483.970,Z 838.065,A 0.000,B 0.000,C 90.000,E1 227.796} C_DIS
LIN {X 0.298,Y -479.904,Z 838.055,A 0.000,B 0.000,C 90.000,E1 225.891} C_DIS
LIN {X -0.011,Y -475.887,Z 838.045,A 0.000,B 0.000,C 90.000,E1 224.069} C_DIS
LIN {X -0.202,Y -470.442,Z 838.031,A 0.000,B 0.000,C 90.000,E1 221.595} C_DIS
LIN {X -0.085,Y -467.191,Z 838.022,A 0.000,B 0.000,C 90.000,E1 220.011} C_DIS
LIN {X 0.036,Y -463.901,Z 838.013,A 0.000,B 0.000,C 90.000,E1 218.418} C_DIS
LIN {X 0.123,Y -460.003,Z 838.003,A 0.000,B 0.000,C 90.000,E1 216.503} C_DIS
LIN {X 0.036,Y -455.216,Z 837.991,A 0.000,B 0.000,C 90.000,E1 214.278} C_DIS
LIN {X 0.112,Y -451.048,Z 837.980,A 0.000,B 0.000,C 90.000,E1 212.339} C_DIS
LIN {X -0.014,Y -449.097,Z 837.974,A 0.000,B 0.000,C 90.000,E1 211.386} C_DIS
LIN {X -0.220,Y -443.082,Z 837.958,A 0.000,B 0.000,C 90.000,E1 208.487} C_DIS
LIN {X 0.002,Y -439.775,Z 837.949,A 0.000,B 0.000,C 90.000,E1 206.821} C_DIS
LIN {X -0.068,Y -437.139,Z 837.942,A 0.000,B 0.000,C 90.000,E1 205.515} C_DIS
LIN {X -0.166,Y -434.486,Z 837.934,A 0.000,B 0.000,C 90.000,E1 204.207} C_DIS
LIN {X 0.117,Y -429.838,Z 837.922,A 0.000,B 0.000,C 90.000,E1 201.844} C_DIS
LIN {X 0.107,Y -426.605,Z 837.912,A 0.000,B 0.000,C 90.000,E1 200.174} C_DIS
LIN {X 0.141,Y -423.299,Z 837.903,A 0.000,B 0.000,C 90.000,E1 198.489} C_DIS
LIN {X 0.054,Y -418.743,Z 837.890,A 0.000,B 0.000,C 90.000,E1 196.134} C_DIS
LIN {X 0.064,Y -416.172,Z 837.882,A 0.000,B 0.000,C 90.000,E1 194.773} C_DIS
LIN {X 0.109,Y -412.038,Z 837.871,A 0.000,B 0.000,C 90.000,E1 192.715} C_DIS
LIN {X 0.053,Y -408.089,Z 837.859,A 0.000,B 0.000,C 90.000,E1 190.658} C_DIS
LIN {X 0.141,Y -404.120,Z 837.848,A 0.000,B 0.000,C 90.000,E1 188.568} C_DIS
LIN {X 0.082,Y -400.734,Z 837.838,A 0.000,B 0.000,C 90.000,E1 186.834} C_DIS
LIN {X -0.087,Y -397.514,Z 837.828,A 0.000,B 0.000,C 90.000,E1 185.106} C_DIS
LIN {X 0.175,Y -392.463,Z 837.811,A 0.000,B 0.000,C 90.000,E1 181.892} C_DIS
LIN {X -0.163,Y -388.160,Z 837.793,A 0.000,B 0.000,C 90.000,E1 178.740} C_DIS
LIN {X 0.060,Y -385.410,Z 837.781,A 0.000,B 0.000,C 90.000,E1 176.560} C_DIS
LIN {X -0.054,Y -383.167,Z 837.771,A 0.000,B 0.000,C 90.000,E1 174.780} C_DIS
LIN {X 0.107,Y -378.856,Z 837.751,A 0.000,B 0.000,C 90.000,E1 171.141} C_DIS
LIN {X -0.147,Y -376.359,Z 837.737,A 0.000,B 0.000,C 90.000,E1 168.634} C_DIS
LIN {X -0.035,Y -374.252,Z 837.723,A 0.000,B 0.000,C 90.000,E1 166.061} C_DIS
LIN {X -0.052,Y -372.711,Z 837.710,A 0.000,B 0.000,C 90.000,E1 163.866} C_DIS
LIN {X 0.145,Y -372.084,Z 837.700,A 0.000,B 0.000,C 90.000,E1 162.000} C_DIS
LIN {X -0.020,Y -372.239,Z 837.690,A 0.000,B 0.000,C 90.000,E1 160.188} C_DIS
LIN {X -0.025,Y -373.009,Z 837.682,A 0.000,B 0.000,C 90.000,E1 158.720} C_DIS
LIN {X 0.079,Y -373.434,Z 837.680,A 0.000,B 0.000,C 90.000,E1 158.337} C_DIS
LIN {X 0.012,Y -374.140,Z 837.676,A 0.000,B 0.000,C 90.000,E1 157.614} C_DIS
LIN {X 0.091,Y -375.123,Z 837.672,A 0.000,B 0.000,C 90.000,E1 156.869} C_DIS
LIN {X -0.111,Y -375.863,Z 837.670,A 0.000,B 0.000,C 90.000,E1 156.538} C_DIS
LIN {X -0.141,Y -376.437,Z 837.668,A 0.000,B 0.000,C 90.000,E1 156.177} C_DIS
LIN {X 0.112,Y -378.305,Z 837.664,A 0.000,B 0.000,C 90.000,E1 155.409} C_DIS
LIN {X 0.086,Y -379.486,Z 837.661,A 0.000,B 0.000,C 90.000,E1 155.049} C_DIS
LIN {X 0.235,Y -380.203,Z 837.661,A 0.000,B 0.000,C 90.000,E1 154.845} C_DIS
LIN {X -0.130,Y -382.040,Z 837.659,A 0.000,B 0.000,C 90.000,E1 154.537} C_DIS
LIN {X 0.021,Y -383.562,Z 837.656,A 0.000,B 0.000,C 90.000,E1 154.152} C_DIS
LIN {X 0.022,Y -386.004,Z 837.654,A 0.000,B 0.000,C 90.000,E1 153.717} C_DIS
LIN {X 0.191,Y -387.205,Z 837.653,A 0.000,B 0.000,C 90.000,E1 153.512} C_DIS
LIN {X -0.125,Y -393.560,Z 837.650,A 0.000,B 0.000,C 90.000,E1 152.922} C_DIS
LIN {X -0.115,Y -400.242,Z 837.647,A 0.000,B 0.000,C 90.000,E1 152.487} C_DIS
LIN {X 0.047,Y -402.142,Z 837.647,A 0.000,B 0.000,C 90.000,E1 152.359} C_DIS
LIN {X 0.042,Y -416.459,Z 837.643,A 0.000,B 0.000,C 90.000,E1 151.769} C_DIS
LIN {X 0.083,Y -426.309,Z 837.641,A 0.000,B 0.000,C 90.000,E1 151.307} C_DIS
LIN {X 0.036,Y -437.481,Z 837.637,A 0.000,B 0.000,C 90.000,E1 150.667} C_DIS
LIN {X 0.044,Y -443.726,Z 837.635,A 0.000,B 0.000,C 90.000,E1 150.255} C_DIS
LIN {X 0.061,Y -449.802,Z 837.632,A 0.000,B 0.000,C 90.000,E1 149.822} C_DIS
LIN {X -0.215,Y -451.303,Z 837.632,A 0.000,B 0.000,C 90.000,E1 149.744} C_DIS
LIN {X 0.062,Y -461.664,Z 837.627,A 0.000,B 0.000,C 90.000,E1 148.820} C_DIS
LIN {X 0.268,Y -468.646,Z 837.623,A 0.000,B 0.000,C 90.000,E1 148.122} C_DIS
LIN {X -0.060,Y -474.306,Z 837.620,A 0.000,B 0.000,C 90.000,E1 147.582} C_DIS
LIN {X 0.014,Y -477.095,Z 837.618,A 0.000,B 0.000,C 90.000,E1 147.296} C_DIS
LIN {X 0.101,Y -482.134,Z 837.615,A 0.000,B 0.000,C 90.000,E1 146.707} C_DIS
LIN {X -0.166,Y -485.709,Z 837.613,A 0.000,B 0.000,C 90.000,E1 146.294} C_DIS
LIN {X 0.007,Y -490.743,Z 837.609,A 0.000,B 0.000,C 90.000,E1 145.674} C_DIS
LIN {X 0.096,Y -495.307,Z 837.606,A 0.000,B 0.000,C 90.000,E1 145.055} C_DIS
LIN {X -0.109,Y -500.383,Z 837.602,A 0.000,B 0.000,C 90.000,E1 144.322} C_DIS
LIN {X -0.059,Y -506.374,Z 837.597,A 0.000,B 0.000,C 90.000,E1 143.417} C_DIS
LIN {X 0.312,Y -513.652,Z 837.590,A 0.000,B 0.000,C 90.000,E1 142.190} C_DIS
LIN {X 0.162,Y -517.292,Z 837.587,A 0.000,B 0.000,C 90.000,E1 141.618} C_DIS
LIN {X 0.307,Y -522.452,Z 837.582,A 0.000,B 0.000,C 90.000,E1 140.723} C_DIS
LIN {X -0.228,Y -527.408,Z 837.577,A 0.000,B 0.000,C 90.000,E1 139.908} C_DIS
LIN {X 0.008,Y -533.773,Z 837.571,A 0.000,B 0.000,C 90.000,E1 138.728} C_DIS
LIN {X -0.101,Y -545.709,Z 837.558,A 0.000,B 0.000,C 90.000,E1 136.458} C_DIS
LIN {X -0.238,Y -550.694,Z 837.553,A 0.000,B 0.000,C 90.000,E1 135.486} C_DIS
LIN {X 0.127,Y -557.269,Z 837.546,A 0.000,B 0.000,C 90.000,E1 134.190} C_DIS
LIN {X 0.034,Y -563.727,Z 837.538,A 0.000,B 0.000,C 90.000,E1 132.813} C_DIS
LIN {X -0.051,Y -570.575,Z 837.530,A 0.000,B 0.000,C 90.000,E1 131.310} C_DIS
LIN {X -0.001,Y -576.944,Z 837.521,A 0.000,B 0.000,C 90.000,E1 129.806} C_DIS
LIN {X -0.272,Y -581.009,Z 837.515,A 0.000,B 0.000,C 90.000,E1 128.749} C_DIS
LIN {X 0.242,Y -584.005,Z 837.511,A 0.000,B 0.000,C 90.000,E1 127.890} C_DIS
LIN {X -0.025,Y -586.575,Z 837.506,A 0.000,B 0.000,C 90.000,E1 127.111} C_DIS
LIN {X 0.284,Y -589.463,Z 837.500,A 0.000,B 0.000,C 90.000,E1 126.011} C_DIS
LIN {X -0.062,Y -591.881,Z 837.494,A 0.000,B 0.000,C 90.000,E1 124.978} C_DIS
LIN {X -0.252,Y -593.481,Z 837.490,A 0.000,B 0.000,C 90.000,E1 124.199} C_DIS
LIN {X 0.174,Y -595.398,Z 837.483,A 0.000,B 0.000,C 90.000,E1 122.832} C_DIS
LIN {X 0.004,Y -596.433,Z 837.478,A 0.000,B 0.000,C 90.000,E1 122.054} C_DIS
LIN {X -0.062,Y -597.338,Z 837.472,A 0.000,B 0.000,C 90.000,E1 121.003} C_DIS
LIN {X -0.020,Y -597.843,Z 837.468,A 0.000,B 0.000,C 90.000,E1 120.207} C_DIS
LIN {X 0.110,Y -598.046,Z 837.465,A 0.000,B 0.000,C 90.000,E1 119.667} C_DIS
LIN {X 0.155,Y -597.972,Z 837.461,A 0.000,B 0.000,C 90.000,E1 118.871} C_DIS
LIN {X -0.089,Y -597.683,Z 837.456,A 0.000,B 0.000,C 90.000,E1 118.103} C_DIS
LIN {X -0.137,Y -597.079,Z 837.450,A 0.000,B 0.000,C 90.000,E1 117.052} C_DIS
LIN {X 0.231,Y -596.616,Z 837.447,A 0.000,B 0.000,C 90.000,E1 116.488} C_DIS
LIN {X -0.108,Y -595.268,Z 837.441,A 0.000,B 0.000,C 90.000,E1 115.463} C_DIS
LIN {X 0.253,Y -594.343,Z 837.439,A 0.000,B 0.000,C 90.000,E1 114.899} C_DIS
LIN {X 0.069,Y -593.211,Z 837.436,A 0.000,B 0.000,C 90.000,E1 114.387} C_DIS
LIN {X -0.026,Y -592.594,Z 837.434,A 0.000,B 0.000,C 90.000,E1 114.131} C_DIS
LIN {X 0.078,Y -590.892,Z 837.431,A 0.000,B 0.000,C 90.000,E1 113.590} C_DIS
LIN {X -0.131,Y -588.883,Z 837.428,A 0.000,B 0.000,C 90.000,E1 113.078} C_DIS
LIN {X -0.186,Y -588.350,Z 837.427,A 0.000,B 0.000,C 90.000,E1 112.950} C_DIS
LIN {X 0.121,Y -585.691,Z 837.424,A 0.000,B 0.000,C 90.000,E1 112.386} C_DIS
LIN {X -0.163,Y -584.645,Z 837.424,A 0.000,B 0.000,C 90.000,E1 112.280} C_DIS
LIN {X -0.272,Y -580.618,Z 837.422,A 0.000,B 0.000,C 90.000,E1 111.897} C_DIS
LIN {X -0.134,Y -577.466,Z 837.420,A 0.000,B 0.000,C 90.000,E1 111.642} C_DIS
LIN {X -0.025,Y -574.381,Z 837.419,A 0.000,B 0.000,C 90.000,E1 111.408} C_DIS
LIN {X 0.171,Y -572.580,Z 837.418,A 0.000,B 0.000,C 90.000,E1 111.280} C_DIS
LIN {X -0.241,Y -570.520,Z 837.418,A 0.000,B 0.000,C 90.000,E1 111.227} C_DIS
LIN {X 0.085,Y -569.131,Z 837.417,A 0.000,B 0.000,C 90.000,E1 111.099} C_DIS
LIN {X 0.178,Y -565.897,Z 837.416,A 0.000,B 0.000,C 90.000,E1 110.791} C_DIS
LIN {X 0.171,Y -565.326,Z 837.415,A 0.000,B 0.000,C 90.000,E1 110.663} C_DIS
LIN {X 0.203,Y -564.305,Z 837.413,A 0.000,B 0.000,C 90.000,E1 110.248} C_DIS
LIN {X 0.090,Y -563.893,Z 837.411,A 0.000,B 0.000,C 90.000,E1 109.939} C_DIS
LIN {X 0.120,Y -563.045,Z 837.409,A 0.000,B 0.000,C 90.000,E1 109.523} C_DIS
LIN {X -0.063,Y -562.319,Z 837.405,A 0.000,B 0.000,C 90.000,E1 108.852} C_DIS
LIN {X -0.230,Y -561.762,Z 837.399,A 0.000,B 0.000,C 90.000,E1 107.764} C_DIS
LIN {X -0.189,Y -562.677,Z 837.372,A 0.000,B 0.000,C 90.000,E1 103.063} C_DIS
LIN {X 0.222,Y -563.726,Z 837.363,A 0.000,B 0.000,C 90.000,E1 101.366} C_DIS
LIN {X -0.225,Y -565.256,Z 837.351,A 0.000,B 0.000,C 90.000,E1 99.208} C_DIS
LIN {X -0.040,Y -566.182,Z 837.343,A 0.000,B 0.000,C 90.000,E1 97.814} C_DIS
LIN {X 0.080,Y -567.073,Z 837.336,A 0.000,B 0.000,C 90.000,E1 96.429} C_DIS
LIN {X -0.249,Y -567.888,Z 837.327,A 0.000,B 0.000,C 90.000,E1 94.816} C_DIS
LIN {X -0.080,Y -568.531,Z 837.318,A 0.000,B 0.000,C 90.000,E1 93.154} C_DIS
LIN {X 0.263,Y -569.157,Z 837.307,A 0.000,B 0.000,C 90.000,E1 91.203} C_DIS
LIN {X -0.239,Y -569.533,Z 837.299,A 0.000,B 0.000,C 90.000,E1 89.885} C_DIS
LIN {X 0.274,Y -569.818,Z 837.293,A 0.000,B 0.000,C 90.000,E1 88.740} C_DIS
LIN {X 0.078,Y -570.206,Z 837.283,A 0.000,B 0.000,C 90.000,E1 86.846} C_DIS
LIN {X -0.103,Y -570.534,Z 837.272,A 0.000,B 0.000,C 90.000,E1 84.951} C_DIS
LIN {X 0.033,Y -570.792,Z 837.264,A 0.000,B 0.000,C 90.000,E1 83.571} C_DIS
LIN {X -0.146,Y -571.164,Z 837.255,A 0.000,B 0.000,C 90.000,E1 81.951} C_DIS
LIN {X 0.151,Y -571.526,Z 837.248,A 0.000,B 0.000,C 90.000,E1 80.557} C_DIS
LIN {X 0.283,Y -572.186,Z 837.237,A 0.000,B 0.000,C 90.000,E1 78.634} C_DIS
LIN {X 0.020,Y -572.620,Z 837.229,A 0.000,B 0.000,C 90.000,E1 77.297} C_DIS
LIN {X -0.156,Y -573.023,Z 837.219,A 0.000,B 0.000,C 90.000,E1 75.408} C_DIS
LIN {X 0.015,Y -573.179,Z 837.214,A 0.000,B 0.000,C 90.000,E1 74.574} C_DIS
LIN {X -0.002,Y -573.285,Z 837.204,A 0.000,B 0.000,C 90.000,E1 72.670} C_DIS
LIN {X -0.034,Y -573.188,Z 837.195,A 0.000,B 0.000,C 90.000,E1 71.040} C_DIS
LIN {X 0.125,Y -573.039,Z 837.186,A 0.000,B 0.000,C 90.000,E1 69.390} C_DIS
LIN {X -0.064,Y -572.926,Z 837.181,A 0.000,B 0.000,C 90.000,E1 68.592} C_DIS
LIN {X 0.105,Y -572.765,Z 837.175,A 0.000,B 0.000,C 90.000,E1 67.486} C_DIS
LIN {X 0.327,Y -572.417,Z 837.167,A 0.000,B 0.000,C 90.000,E1 66.102} C_DIS
LIN {X 0.137,Y -571.779,Z 837.158,A 0.000,B 0.000,C 90.000,E1 64.485} C_DIS
LIN {X 0.073,Y -571.198,Z 837.151,A 0.000,B 0.000,C 90.000,E1 63.127} C_DIS
LIN {X -0.162,Y -570.456,Z 837.142,A 0.000,B 0.000,C 90.000,E1 61.513} C_DIS
LIN {X 0.270,Y -570.146,Z 837.139,A 0.000,B 0.000,C 90.000,E1 60.923} C_DIS
LIN {X 0.031,Y -569.473,Z 837.134,A 0.000,B 0.000,C 90.000,E1 60.127} C_DIS
LIN {X 0.204,Y -568.120,Z 837.127,A 0.000,B 0.000,C 90.000,E1 58.742} C_DIS
LIN {X 0.162,Y -566.515,Z 837.119,A 0.000,B 0.000,C 90.000,E1 57.375} C_DIS
LIN {X -0.014,Y -564.982,Z 837.113,A 0.000,B 0.000,C 90.000,E1 56.294} C_DIS
LIN {X -0.008,Y -563.670,Z 837.108,A 0.000,B 0.000,C 90.000,E1 55.468} C_DIS
LIN {X -0.018,Y -562.217,Z 837.104,A 0.000,B 0.000,C 90.000,E1 54.642} C_DIS
LIN {X -0.172,Y -560.609,Z 837.099,A 0.000,B 0.000,C 90.000,E1 53.829} C_DIS
LIN {X -0.131,Y -558.145,Z 837.093,A 0.000,B 0.000,C 90.000,E1 52.718} C_DIS
LIN {X -0.315,Y -556.019,Z 837.088,A 0.000,B 0.000,C 90.000,E1 51.904} C_DIS
LIN {X -0.158,Y -554.494,Z 837.085,A 0.000,B 0.000,C 90.000,E1 51.331} C_DIS
LIN {X -0.026,Y -551.928,Z 837.081,A 0.000,B 0.000,C 90.000,E1 50.481} C_DIS
LIN {X 0.097,Y -550.094,Z 837.077,A 0.000,B 0.000,C 90.000,E1 49.908} C_DIS
LIN {X -0.169,Y -546.963,Z 837.073,A 0.000,B 0.000,C 90.000,E1 49.094} C_DIS
LIN {X 0.056,Y -544.096,Z 837.069,A 0.000,B 0.000,C 90.000,E1 48.366} C_DIS
LIN {X 0.106,Y -541.644,Z 837.066,A 0.000,B 0.000,C 90.000,E1 47.796} C_DIS
LIN {X -0.083,Y -538.187,Z 837.062,A 0.000,B 0.000,C 90.000,E1 47.106} C_DIS
LIN {X -0.116,Y -535.226,Z 837.059,A 0.000,B 0.000,C 90.000,E1 46.539} C_DIS
LIN {X -0.166,Y -531.981,Z 837.055,A 0.000,B 0.000,C 90.000,E1 45.972} C_DIS
LIN {X -0.073,Y -527.334,Z 837.051,A 0.000,B 0.000,C 90.000,E1 45.243} C_DIS
LIN {X -0.014,Y -523.493,Z 837.048,A 0.000,B 0.000,C 90.000,E1 44.676} C_DIS
LIN {X -0.100,Y -519.168,Z 837.045,A 0.000,B 0.000,C 90.000,E1 44.109} C_DIS
LIN {X -0.156,Y -514.582,Z 837.042,A 0.000,B 0.000,C 90.000,E1 43.542} C_DIS
LIN {X 0.024,Y -511.081,Z 837.039,A 0.000,B 0.000,C 90.000,E1 43.095} C_DIS
LIN {X -0.309,Y -507.188,Z 837.037,A 0.000,B 0.000,C 90.000,E1 42.690} C_DIS
LIN {X 0.152,Y -500.390,Z 837.033,A 0.000,B 0.000,C 90.000,E1 41.919} C_DIS
LIN {X 0.001,Y -497.900,Z 837.032,A 0.000,B 0.000,C 90.000,E1 41.676} C_DIS
LIN {X -0.011,Y -490.624,Z 837.028,A 0.000,B 0.000,C 90.000,E1 40.987} C_DIS
LIN {X -0.291,Y -486.120,Z 837.026,A 0.000,B 0.000,C 90.000,E1 40.620} C_DIS
LIN {X 0.204,Y -478.586,Z 837.022,A 0.000,B 0.000,C 90.000,E1 39.930} C_DIS
LIN {X 0.151,Y -469.248,Z 837.018,A 0.000,B 0.000,C 90.000,E1 39.197} C_DIS
LIN {X 0.020,Y -458.255,Z 837.013,A 0.000,B 0.000,C 90.000,E1 38.382} C_DIS
LIN {X -0.118,Y -447.177,Z 837.009,A 0.000,B 0.000,C 90.000,E1 37.569} C_DIS
LIN {X 0.100,Y -428.242,Z 837.001,A 0.000,B 0.000,C 90.000,E1 36.091} C_DIS
LIN {X 0.027,Y -414.350,Z 836.994,A 0.000,B 0.000,C 90.000,E1 34.945} C_DIS
LIN {X 0.106,Y -404.102,Z 836.989,A 0.000,B 0.000,C 90.000,E1 33.992} C_DIS
LIN {X 0.057,Y -400.214,Z 836.987,A 0.000,B 0.000,C 90.000,E1 33.579} C_DIS
LIN {X 0.029,Y -395.846,Z 836.983,A 0.000,B 0.000,C 90.000,E1 33.007} C_DIS
LIN {X 0.025,Y -395.223,Z 836.982,A 0.000,B 0.000,C 90.000,E1 32.832} C_DIS
LIN {X -0.095,Y -393.837,Z 836.977,A 0.000,B 0.000,C 90.000,E1 31.878} C_DIS
LIN {X -0.108,Y -391.123,Z 836.969,A 0.000,B 0.000,C 90.000,E1 30.463} C_DIS
LIN {X -0.208,Y -391.317,Z 836.963,A 0.000,B 0.000,C 90.000,E1 29.411} C_DIS
LIN {X 0.141,Y -392.715,Z 836.949,A 0.000,B 0.000,C 90.000,E1 26.873} C_DIS
LIN {X -0.141,Y -394.666,Z 836.934,A 0.000,B 0.000,C 90.000,E1 24.079} C_DIS
LIN {X -0.081,Y -396.374,Z 836.922,A 0.000,B 0.000,C 90.000,E1 21.950} C_DIS
LIN {X -0.061,Y -399.265,Z 836.904,A 0.000,B 0.000,C 90.000,E1 18.779} C_DIS
LIN {X 0.017,Y -402.008,Z 836.891,A 0.000,B 0.000,C 90.000,E1 16.315} C_DIS
LIN {X 0.046,Y -406.323,Z 836.873,A 0.000,B 0.000,C 90.000,E1 13.175} C_DIS
LIN {X -0.068,Y -410.709,Z 836.858,A 0.000,B 0.000,C 90.000,E1 10.423} C_DIS
LIN {X 0.090,Y -413.633,Z 836.848,A 0.000,B 0.000,C 90.000,E1 8.681} C_DIS
LIN {X -0.165,Y -417.270,Z 836.837,A 0.000,B 0.000,C 90.000,E1 6.663} C_DIS
LIN {X 0.209,Y -422.913,Z 836.820,A 0.000,B 0.000,C 90.000,E1 3.555} C_DIS
LIN {X -0.070,Y -429.897,Z 836.801,A 0.000,B 0.000,C 90.000,E1 0.229} C_DIS
LIN {X 0.150,Y -434.728,Z 836.790,A 0.000,B 0.000,C 90.000,E1 358.108} C_DIS
LIN {X 0.015,Y -440.313,Z 836.777,A 0.000,B 0.000,C 90.000,E1 355.812} C_DIS
LIN {X 0.050,Y -446.179,Z 836.764,A 0.000,B 0.000,C 90.000,E1 353.514} C_DIS
LIN {X 0.080,Y -448.895,Z 836.759,A 0.000,B 0.000,C 90.000,E1 352.534} C_DIS
LIN {X -0.007,Y -450.567,Z 836.756,A 0.000,B 0.000,C 90.000,E1 352.064} C_DIS
LIN {X -0.192,Y -452.714,Z 836.753,A 0.000,B 0.000,C 90.000,E1 351.602} C_DIS
LIN {X -0.018,Y -454.995,Z 836.751,A 0.000,B 0.000,C 90.000,E1 351.197} C_DIS
LIN {X -0.106,Y -459.095,Z 836.749,A 0.000,B 0.000,C 90.000,E1 350.792} C_DIS
LIN {X -0.052,Y -462.809,Z 836.747,A 0.000,B 0.000,C 90.000,E1 350.500} C_DIS
LIN {X -0.074,Y -466.098,Z 836.746,A 0.000,B 0.000,C 90.000,E1 350.274} C_DIS
LIN {X -0.226,Y -481.420,Z 836.741,A 0.000,B 0.000,C 90.000,E1 349.398} C_DIS
LIN {X 0.228,Y -489.535,Z 836.738,A 0.000,B 0.000,C 90.000,E1 348.870} C_DIS
LIN {X 0.038,Y -499.058,Z 836.735,A 0.000,B 0.000,C 90.000,E1 348.285} C_DIS
LIN {X 0.187,Y -508.549,Z 836.732,A 0.000,B 0.000,C 90.000,E1 347.645} C_DIS
LIN {X 0.276,Y -517.926,Z 836.728,A 0.000,B 0.000,C 90.000,E1 346.992} C_DIS
LIN {X 0.280,Y -528.731,Z 836.724,A 0.000,B 0.000,C 90.000,E1 346.228} C_DIS
LIN {X -0.027,Y -536.174,Z 836.721,A 0.000,B 0.000,C 90.000,E1 345.700} C_DIS
LIN {X 0.091,Y -543.407,Z 836.717,A 0.000,B 0.000,C 90.000,E1 345.102} C_DIS
LIN {X 0.049,Y -549.136,Z 836.715,A 0.000,B 0.000,C 90.000,E1 344.629} C_DIS
LIN {X -0.241,Y -557.381,Z 836.711,A 0.000,B 0.000,C 90.000,E1 343.921} C_DIS
LIN {X 0.159,Y -561.298,Z 836.708,A 0.000,B 0.000,C 90.000,E1 343.504} C_DIS
LIN {X 0.306,Y -566.459,Z 836.706,A 0.000,B 0.000,C 90.000,E1 342.960} C_DIS
LIN {X -0.184,Y -571.428,Z 836.703,A 0.000,B 0.000,C 90.000,E1 342.472} C_DIS
LIN {X 0.072,Y -577.371,Z 836.699,A 0.000,B 0.000,C 90.000,E1 341.764} C_DIS
LIN {X 0.091,Y -581.788,Z 836.696,A 0.000,B 0.000,C 90.000,E1 341.221} C_DIS
LIN {X 0.068,Y -586.832,Z 836.692,A 0.000,B 0.000,C 90.000,E1 340.550} C_DIS
LIN {X 0.154,Y -590.773,Z 836.689,A 0.000,B 0.000,C 90.000,E1 340.007} C_DIS
LIN {X 0.156,Y -596.028,Z 836.685,A 0.000,B 0.000,C 90.000,E1 339.209} C_DIS
LIN {X 0.213,Y -600.972,Z 836.680,A 0.000,B 0.000,C 90.000,E1 338.411} C_DIS
LIN {X -0.205,Y -604.848,Z 836.677,A 0.000,B 0.000,C 90.000,E1 337.794} C_DIS
LIN {X -0.114,Y -610.805,Z 836.671,A 0.000,B 0.000,C 90.000,E1 336.741} C_DIS
LIN {X 0.319,Y -615.790,Z 836.666,A 0.000,B 0.000,C 90.000,E1 335.793} C_DIS
LIN {X -0.006,Y -621.171,Z 836.660,A 0.000,B 0.000,C 90.000,E1 334.793} C_DIS
LIN {X -0.008,Y -624.989,Z 836.656,A 0.000,B 0.000,C 90.000,E1 334.024} C_DIS
LIN {X 0.032,Y -628.644,Z 836.651,A 0.000,B 0.000,C 90.000,E1 333.256} C_DIS
LIN {X 0.134,Y -633.184,Z 836.646,A 0.000,B 0.000,C 90.000,E1 332.231} C_DIS
LIN {X -0.270,Y -637.493,Z 836.640,A 0.000,B 0.000,C 90.000,E1 331.257} C_DIS
LIN {X 0.249,Y -641.614,Z 836.635,A 0.000,B 0.000,C 90.000,E1 330.205} C_DIS
LIN {X 0.271,Y -645.512,Z 836.629,A 0.000,B 0.000,C 90.000,E1 329.203} C_DIS
LIN {X -0.205,Y -649.053,Z 836.624,A 0.000,B 0.000,C 90.000,E1 328.250} C_DIS
LIN {X -0.002,Y -653.229,Z 836.617,A 0.000,B 0.000,C 90.000,E1 326.993} C_DIS
LIN {X 0.433,Y -655.515,Z 836.613,A 0.000,B 0.000,C 90.000,E1 326.215} C_DIS
LIN {X 0.078,Y -658.382,Z 836.607,A 0.000,B 0.000,C 90.000,E1 325.261} C_DIS
LIN {X 0.076,Y -661.659,Z 836.600,A 0.000,B 0.000,C 90.000,E1 324.036} C_DIS
LIN {X 0.123,Y -662.866,Z 836.598,A 0.000,B 0.000,C 90.000,E1 323.543} C_DIS
LIN {X -0.201,Y -665.496,Z 836.591,A 0.000,B 0.000,C 90.000,E1 322.351} C_DIS
LIN {X -0.177,Y -667.416,Z 836.585,A 0.000,B 0.000,C 90.000,E1 321.376} C_DIS
LIN {X 0.397,Y -669.129,Z 836.580,A 0.000,B 0.000,C 90.000,E1 320.356} C_DIS
LIN {X 0.045,Y -671.051,Z 836.573,A 0.000,B 0.000,C 90.000,E1 319.175} C_DIS
LIN {X 0.188,Y -673.656,Z 836.564,A 0.000,B 0.000,C 90.000,E1 317.472} C_DIS
LIN {X -0.208,Y -674.694,Z 836.560,A 0.000,B 0.000,C 90.000,E1 316.782} C_DIS
LIN {X -0.008,Y -676.801,Z 836.550,A 0.000,B 0.000,C 90.000,E1 315.081} C_DIS
LIN {X 0.131,Y -677.920,Z 836.545,A 0.000,B 0.000,C 90.000,E1 314.109} C_DIS
LIN {X -0.067,Y -679.691,Z 836.536,A 0.000,B 0.000,C 90.000,E1 312.447} C_DIS
LIN {X 0.227,Y -681.217,Z 836.528,A 0.000,B 0.000,C 90.000,E1 310.987} C_DIS
LIN {X 0.104,Y -682.601,Z 836.520,A 0.000,B 0.000,C 90.000,E1 309.564} C_DIS
LIN {X 0.150,Y -684.075,Z 836.511,A 0.000,B 0.000,C 90.000,E1 307.890} C_DIS
LIN {X 0.198,Y -685.302,Z 836.503,A 0.000,B 0.000,C 90.000,E1 306.457} C_DIS
LIN {X -0.320,Y -686.282,Z 836.496,A 0.000,B 0.000,C 90.000,E1 305.311} C_DIS
LIN {X -0.071,Y -687.276,Z 836.488,A 0.000,B 0.000,C 90.000,E1 303.865} C_DIS
LIN {X -0.166,Y -688.414,Z 836.479,A 0.000,B 0.000,C 90.000,E1 302.212} C_DIS
LIN {X -0.248,Y -689.472,Z 836.471,A 0.000,B 0.000,C 90.000,E1 300.797} C_DIS
LIN {X 0.141,Y -690.899,Z 836.461,A 0.000,B 0.000,C 90.000,E1 298.871} C_DIS
LIN {X 0.030,Y -692.044,Z 836.453,A 0.000,B 0.000,C 90.000,E1 297.462} C_DIS
LIN {X -0.176,Y -693.669,Z 836.442,A 0.000,B 0.000,C 90.000,E1 295.591} C_DIS
LIN {X 0.142,Y -694.688,Z 836.436,A 0.000,B 0.000,C 90.000,E1 294.387} C_DIS
LIN {X -0.279,Y -694.794,Z 836.433,A 0.000,B 0.000,C 90.000,E1 293.951} C_DIS
LIN {X -0.030,Y -694.743,Z 836.432,A 0.000,B 0.000,C 90.000,E1 293.695} C_DIS
LIN {X 0.189,Y -694.120,Z 836.429,A 0.000,B 0.000,C 90.000,E1 293.206} C_DIS
LIN {X -0.203,Y -693.453,Z 836.428,A 0.000,B 0.000,C 90.000,E1 293.003} C_DIS
LIN {X 0.008,Y -690.861,Z 836.425,A 0.000,B 0.000,C 90.000,E1 292.514} C_DIS
LIN {X 0.124,Y -690.115,Z 836.424,A 0.000,B 0.000,C 90.000,E1 292.386} C_DIS
LIN {X -0.022,Y -689.012,Z 836.424,A 0.000,B 0.000,C 90.000,E1 292.280} C_DIS
LIN {X 0.205,Y -685.670,Z 836.422,A 0.000,B 0.000,C 90.000,E1 292.025} C_DIS
LIN {X 0.055,Y -682.818,Z 836.421,A 0.000,B 0.000,C 90.000,E1 291.844} C_DIS
LIN {X -0.212,Y -681.110,Z 836.421,A 0.000,B 0.000,C 90.000,E1 291.770} C_DIS
LIN {X 0.097,Y -676.294,Z 836.420,A 0.000,B 0.000,C 90.000,E1 291.589} C_DIS
LIN {X 0.323,Y -670.983,Z 836.419,A 0.000,B 0.000,C 90.000,E1 291.408} C_DIS
LIN {X 0.131,Y -664.010,Z 836.418,A 0.000,B 0.000,C 90.000,E1 291.280} C_DIS
LIN {X -0.185,Y -654.732,Z 836.417,A 0.000,B 0.000,C 90.000,E1 291.153} C_DIS
LIN {X 0.210,Y -645.403,Z 836.416,A 0.000,B 0.000,C 90.000,E1 290.918} C_DIS
LIN {X -0.179,Y -639.615,Z 836.415,A 0.000,B 0.000,C 90.000,E1 290.791} C_DIS
LIN {X 0.303,Y -637.298,Z 836.415,A 0.000,B 0.000,C 90.000,E1 290.663} C_DIS
LIN {X 0.116,Y -633.427,Z 836.414,A 0.000,B 0.000,C 90.000,E1 290.556} C_DIS
LIN {X 0.093,Y -627.154,Z 836.413,A 0.000,B 0.000,C 90.000,E1 290.248} C_DIS
LIN {X 0.026,Y -625.686,Z 836.412,A 0.000,B 0.000,C 90.000,E1 290.120} C_DIS
LIN {X -0.015,Y -625.678,Z 836.412,A 0.000,B 0.000,C 90.000,E1 290.120} C_DIS
LIN {X -0.019,Y -625.393,Z 836.410,A 0.000,B 0.000,C 90.000,E1 289.866} C_DIS
LIN {X 0.242,Y -626.996,Z 836.408,A 0.000,B 0.000,C 90.000,E1 289.396} C_DIS
LIN {X -0.104,Y -630.926,Z 836.404,A 0.000,B 0.000,C 90.000,E1 288.725} C_DIS
LIN {X 0.164,Y -635.186,Z 836.400,A 0.000,B 0.000,C 90.000,E1 287.946} C_DIS
LIN {X -0.183,Y -638.762,Z 836.396,A 0.000,B 0.000,C 90.000,E1 287.221} C_DIS
LIN {X 0.275,Y -640.956,Z 836.393,A 0.000,B 0.000,C 90.000,E1 286.677} C_DIS
LIN {X -0.206,Y -643.752,Z 836.389,A 0.000,B 0.000,C 90.000,E1 285.969} C_DIS
LIN {X 0.285,Y -645.363,Z 836.386,A 0.000,B 0.000,C 90.000,E1 285.426} C_DIS
LIN {X -0.008,Y -646.712,Z 836.383,A 0.000,B 0.000,C 90.000,E1 284.954} C_DIS
LIN {X 0.198,Y -648.381,Z 836.379,A 0.000,B 0.000,C 90.000,E1 284.189} C_DIS
LIN {X 0.082,Y -649.324,Z 836.376,A 0.000,B 0.000,C 90.000,E1 283.703} C_DIS
LIN {X -0.188,Y -649.856,Z 836.373,A 0.000,B 0.000,C 90.000,E1 283.231} C_DIS
LIN {X 0.036,Y -650.214,Z 836.371,A 0.000,B 0.000,C 90.000,E1 282.715} C_DIS
LIN {X 0.281,Y -650.284,Z 836.367,A 0.000,B 0.000,C 90.000,E1 281.951} C_DIS
LIN {X -0.115,Y -649.943,Z 836.362,A 0.000,B 0.000,C 90.000,E1 281.243} C_DIS
LIN {X 0.133,Y -649.324,Z 836.360,A 0.000,B 0.000,C 90.000,E1 280.725} C_DIS
LIN {X -0.280,Y -647.938,Z 836.356,A 0.000,B 0.000,C 90.000,E1 280.018} C_DIS
LIN {X -0.039,Y -646.716,Z 836.353,A 0.000,B 0.000,C 90.000,E1 279.500} C_DIS
LIN {X 0.302,Y -645.083,Z 836.350,A 0.000,B 0.000,C 90.000,E1 278.973} C_DIS
LIN {X -0.236,Y -642.397,Z 836.347,A 0.000,B 0.000,C 90.000,E1 278.398} C_DIS
LIN {X 0.064,Y -639.817,Z 836.344,A 0.000,B 0.000,C 90.000,E1 277.871} C_DIS
LIN {X 0.120,Y -635.956,Z 836.340,A 0.000,B 0.000,C 90.000,E1 277.239} C_DIS
LIN {X 0.286,Y -632.283,Z 836.338,A 0.000,B 0.000,C 90.000,E1 276.720} C_DIS
LIN {X -0.199,Y -627.999,Z 836.335,A 0.000,B 0.000,C 90.000,E1 276.258} C_DIS
LIN {X 0.282,Y -626.758,Z 836.334,A 0.000,B 0.000,C 90.000,E1 276.087} C_DIS
LIN {X 0.099,Y -621.316,Z 836.331,A 0.000,B 0.000,C 90.000,E1 275.625} C_DIS
LIN {X -0.285,Y -615.363,Z 836.329,A 0.000,B 0.000,C 90.000,E1 275.220} C_DIS
LIN {X -0.054,Y -612.158,Z 836.328,A 0.000,B 0.000,C 90.000,E1 274.992} C_DIS
LIN {X -0.228,Y -605.515,Z 836.326,A 0.000,B 0.000,C 90.000,E1 274.645} C_DIS
LIN {X -0.008,Y -598.584,Z 836.324,A 0.000,B 0.000,C 90.000,E1 274.302} C_DIS
LIN {X -0.051,Y -591.647,Z 836.322,A 0.000,B 0.000,C 90.000,E1 274.012} C_DIS
LIN {X 0.169,Y -584.507,Z 836.321,A 0.000,B 0.000,C 90.000,E1 273.726} C_DIS
LIN {X 0.248,Y -578.819,Z 836.320,A 0.000,B 0.000,C 90.000,E1 273.555} C_DIS
LIN {X 0.014,Y -571.689,Z 836.319,A 0.000,B 0.000,C 90.000,E1 273.440} C_DIS
LIN {X 0.043,Y -565.844,Z 836.319,A 0.000,B 0.000,C 90.000,E1 273.383} C_DIS
LIN {X 0.150,Y -554.255,Z 836.319,A 0.000,B 0.000,C 90.000,E1 273.326} C_DIS
LIN {X -0.025,Y -553.169,Z 836.319,A 0.000,B 0.000,C 90.000,E1 273.326} C_DIS
LIN {X 0.201,Y -550.630,Z 836.318,A 0.000,B 0.000,C 90.000,E1 273.212} C_DIS
LIN {X 0.163,Y -550.566,Z 836.318,A 0.000,B 0.000,C 90.000,E1 273.212} C_DIS
LIN {X -0.033,Y -549.593,Z 836.317,A 0.000,B 0.000,C 90.000,E1 273.037} C_DIS
LIN {X -0.229,Y -548.592,Z 836.315,A 0.000,B 0.000,C 90.000,E1 272.636} C_DIS
LIN {X -0.016,Y -547.192,Z 836.308,A 0.000,B 0.000,C 90.000,E1 271.489} C_DIS
LIN {X -0.141,Y -544.986,Z 836.293,A 0.000,B 0.000,C 90.000,E1 268.682} C_DIS
LIN {X 0.084,Y -543.814,Z 836.283,A 0.000,B 0.000,C 90.000,E1 266.963} C_DIS
LIN {X -0.233,Y -542.658,Z 836.274,A 0.000,B 0.000,C 90.000,E1 265.298} C_DIS
LIN {X 0.002,Y -541.732,Z 836.266,A 0.000,B 0.000,C 90.000,E1 263.856} C_DIS
LIN {X 0.087,Y -541.032,Z 836.261,A 0.000,B 0.000,C 90.000,E1 262.996} C_DIS
LIN {X -0.099,Y -539.488,Z 836.252,A 0.000,B 0.000,C 90.000,E1 261.310} C_DIS
LIN {X 0.162,Y -538.159,Z 836.244,A 0.000,B 0.000,C 90.000,E1 259.859} C_DIS
LIN {X -0.081,Y -536.413,Z 836.234,A 0.000,B 0.000,C 90.000,E1 258.173} C_DIS
LIN {X -0.142,Y -534.690,Z 836.225,A 0.000,B 0.000,C 90.000,E1 256.464} C_DIS
LIN {X -0.039,Y -534.077,Z 836.222,A 0.000,B 0.000,C 90.000,E1 255.880} C_DIS
LIN {X -0.020,Y -532.037,Z 836.212,A 0.000,B 0.000,C 90.000,E1 254.157} C_DIS
LIN {X 0.109,Y -530.022,Z 836.202,A 0.000,B 0.000,C 90.000,E1 252.417} C_DIS
LIN {X 0.001,Y -528.627,Z 836.196,A 0.000,B 0.000,C 90.000,E1 251.275} C_DIS
LIN {X 0.044,Y -527.076,Z 836.190,A 0.000,B 0.000,C 90.000,E1 250.115} C_DIS
LIN {X -0.273,Y -524.651,Z 836.180,A 0.000,B 0.000,C 90.000,E1 248.411} C_DIS
LIN {X 0.221,Y -522.175,Z 836.170,A 0.000,B 0.000,C 90.000,E1 246.613} C_DIS
LIN {X -0.120,Y -520.390,Z 836.164,A 0.000,B 0.000,C 90.000,E1 245.485} C_DIS
LIN {X 0.203,Y -518.572,Z 836.157,A 0.000,B 0.000,C 90.000,E1 244.280} C_DIS
LIN {X 0.033,Y -516.585,Z 836.151,A 0.000,B 0.000,C 90.000,E1 243.127} C_DIS
LIN {X 0.190,Y -512.934,Z 836.139,A 0.000,B 0.000,C 90.000,E1 241.051} C_DIS
LIN {X 0.156,Y -509.685,Z 836.130,A 0.000,B 0.000,C 90.000,E1 239.282} C_DIS
LIN {X 0.244,Y -506.863,Z 836.121,A 0.000,B 0.000,C 90.000,E1 237.788} C_DIS
LIN {X 0.079,Y -505.071,Z 836.116,A 0.000,B 0.000,C 90.000,E1 236.914} C_DIS
LIN {X 0.058,Y -502.509,Z 836.110,A 0.000,B 0.000,C 90.000,E1 235.722} C_DIS
LIN {X 0.006,Y -499.787,Z 836.103,A 0.000,B 0.000,C 90.000,E1 234.529} C_DIS
LIN {X -0.094,Y -494.770,Z 836.091,A 0.000,B 0.000,C 90.000,E1 232.431} C_DIS
LIN {X -0.215,Y -492.694,Z 836.086,A 0.000,B 0.000,C 90.000,E1 231.537} C_DIS
LIN {X 0.027,Y -490.537,Z 836.081,A 0.000,B 0.000,C 90.000,E1 230.598} C_DIS
LIN {X -0.157,Y -487.081,Z 836.073,A 0.000,B 0.000,C 90.000,E1 229.094} C_DIS
LIN {X -0.082,Y -483.472,Z 836.064,A 0.000,B 0.000,C 90.000,E1 227.553} C_DIS
LIN {X -0.301,Y -479.361,Z 836.054,A 0.000,B 0.000,C 90.000,E1 225.729} C_DIS
LIN {X 0.289,Y -476.081,Z 836.045,A 0.000,B 0.000,C 90.000,E1 224.109} C_DIS
LIN {X 0.034,Y -473.258,Z 836.038,A 0.000,B 0.000,C 90.000,E1 222.894} C_DIS
LIN {X -0.030,Y -469.357,Z 836.028,A 0.000,B 0.000,C 90.000,E1 221.024} C_DIS
LIN {X 0.072,Y -466.077,Z 836.019,A 0.000,B 0.000,C 90.000,E1 219.439} C_DIS
LIN {X -0.009,Y -460.841,Z 836.005,A 0.000,B 0.000,C 90.000,E1 216.916} C_DIS
LIN {X -0.028,Y -458.104,Z 835.998,A 0.000,B 0.000,C 90.000,E1 215.644} C_DIS
LIN {X 0.011,Y -454.735,Z 835.989,A 0.000,B 0.000,C 90.000,E1 214.040} C_DIS
LIN {X -0.008,Y -449.315,Z 835.975,A 0.000,B 0.000,C 90.000,E1 211.465} C_DIS
LIN {X -0.043,Y -443.932,Z 835.960,A 0.000,B 0.000,C 90.000,E1 208.871} C_DIS
LIN {X -0.201,Y -440.663,Z 835.951,A 0.000,B 0.000,C 90.000,E1 207.257} C_DIS
LIN {X -0.029,Y -437.358,Z 835.942,A 0.000,B 0.000,C 90.000,E1 205.591} C_DIS
LIN {X 0.059,Y -434.726,Z 835.935,A 0.000,B 0.000,C 90.000,E1 204.259} C_DIS
LIN {X -0.058,Y -430.075,Z 835.922,A 0.000,B 0.000,C 90.000,E1 201.950} C_DIS
LIN {X 0.181,Y -426.854,Z 835.913,A 0.000,B 0.000,C 90.000,E1 200.248} C_DIS
LIN {X -0.040,Y -423.534,Z 835.903,A 0.000,B 0.000,C 90.000,E1 198.598} C_DIS
LIN {X -0.079,Y -418.350,Z 835.888,A 0.000,B 0.000,C 90.000,E1 195.898} C_DIS
LIN {X -0.074,Y -415.748,Z 835.881,A 0.000,B 0.000,C 90.000,E1 194.537} C_DIS
LIN {X -0.074,Y -412.328,Z 835.871,A 0.000,B 0.000,C 90.000,E1 192.827} C_DIS
LIN {X -0.203,Y -408.366,Z 835.860,A 0.000,B 0.000,C 90.000,E1 190.782} C_DIS
LIN {X -0.035,Y -404.400,Z 835.848,A 0.000,B 0.000,C 90.000,E1 188.681} C_DIS
LIN {X -0.090,Y -401.055,Z 835.839,A 0.000,B 0.000,C 90.000,E1 186.947} C_DIS
LIN {X 0.142,Y -397.826,Z 835.829,A 0.000,B 0.000,C 90.000,E1 185.163} C_DIS
LIN {X 0.018,Y -392.749,Z 835.811,A 0.000,B 0.000,C 90.000,E1 182.007} C_DIS
LIN {X 0.081,Y -388.420,Z 835.793,A 0.000,B 0.000,C 90.000,E1 178.797} C_DIS
LIN {X -0.075,Y -385.721,Z 835.781,A 0.000,B 0.000,C 90.000,E1 176.674} C_DIS
LIN {X -0.181,Y -383.478,Z 835.772,A 0.000,B 0.000,C 90.000,E1 174.894} C_DIS
LIN {X 0.001,Y -379.190,Z 835.751,A 0.000,B 0.000,C 90.000,E1 171.254} C_DIS
LIN {X 0.058,Y -376.717,Z 835.737,A 0.000,B 0.000,C 90.000,E1 168.701} C_DIS
LIN {X -0.135,Y -374.267,Z 835.721,A 0.000,B 0.000,C 90.000,E1 165.811} C_DIS
LIN {X -0.110,Y -372.999,Z 835.711,A 0.000,B 0.000,C 90.000,E1 163.976} C_DIS
LIN {X -0.015,Y -372.221,Z 835.701,A 0.000,B 0.000,C 90.000,E1 162.127} C_DIS
LIN {X -0.088,Y -372.316,Z 835.688,A 0.000,B 0.000,C 90.000,E1 159.934} C_DIS
LIN {X -0.054,Y -372.750,Z 835.682,A 0.000,B 0.000,C 90.000,E1 158.827} C_DIS
LIN {X -0.014,Y -373.635,Z 835.676,A 0.000,B 0.000,C 90.000,E1 157.720} C_DIS
LIN {X 0.064,Y -374.422,Z 835.672,A 0.000,B 0.000,C 90.000,E1 156.975} C_DIS
LIN {X 0.040,Y -375.102,Z 835.670,A 0.000,B 0.000,C 90.000,E1 156.613} C_DIS
LIN {X 0.158,Y -375.625,Z 835.668,A 0.000,B 0.000,C 90.000,E1 156.230} C_DIS
LIN {X -0.094,Y -377.112,Z 835.664,A 0.000,B 0.000,C 90.000,E1 155.537} C_DIS
LIN {X 0.035,Y -377.980,Z 835.662,A 0.000,B 0.000,C 90.000,E1 155.153} C_DIS
LIN {X 0.144,Y -380.195,Z 835.658,A 0.000,B 0.000,C 90.000,E1 154.409} C_DIS
LIN {X -0.066,Y -382.372,Z 835.655,A 0.000,B 0.000,C 90.000,E1 153.896} C_DIS
LIN {X 0.079,Y -385.176,Z 835.652,A 0.000,B 0.000,C 90.000,E1 153.332} C_DIS
LIN {X 0.075,Y -388.843,Z 835.649,A 0.000,B 0.000,C 90.000,E1 152.794} C_DIS
LIN {X 0.017,Y -395.729,Z 835.645,A 0.000,B 0.000,C 90.000,E1 152.153} C_DIS
LIN {X -0.023,Y -397.414,Z 835.645,A 0.000,B 0.000,C 90.000,E1 152.025} C_DIS
LIN {X 0.144,Y -401.274,Z 835.643,A 0.000,B 0.000,C 90.000,E1 151.769} C_DIS
LIN {X 0.060,Y -404.861,Z 835.642,A 0.000,B 0.000,C 90.000,E1 151.591} C_DIS
LIN {X -0.103,Y -417.333,Z 835.639,A 0.000,B 0.000,C 90.000,E1 151.101} C_DIS
LIN {X -0.134,Y -424.279,Z 835.638,A 0.000,B 0.000,C 90.000,E1 150.795} C_DIS
LIN {X -0.156,Y -430.724,Z 835.636,A 0.000,B 0.000,C 90.000,E1 150.461} C_DIS
LIN {X 0.063,Y -433.817,Z 835.635,A 0.000,B 0.000,C 90.000,E1 150.255} C_DIS
LIN {X 0.175,Y -446.655,Z 835.630,A 0.000,B 0.000,C 90.000,E1 149.410} C_DIS
LIN {X -0.210,Y -452.348,Z 835.628,A 0.000,B 0.000,C 90.000,E1 148.997} C_DIS
LIN {X 0.006,Y -459.952,Z 835.624,A 0.000,B 0.000,C 90.000,E1 148.329} C_DIS
LIN {X -0.039,Y -464.327,Z 835.622,A 0.000,B 0.000,C 90.000,E1 147.946} C_DIS
LIN {X -0.020,Y -476.344,Z 835.615,A 0.000,B 0.000,C 90.000,E1 146.707} C_DIS
LIN {X 0.040,Y -478.993,Z 835.614,A 0.000,B 0.000,C 90.000,E1 146.421} C_DIS
LIN {X -0.037,Y -485.235,Z 835.609,A 0.000,B 0.000,C 90.000,E1 145.674} C_DIS
LIN {X -0.150,Y -487.793,Z 835.608,A 0.000,B 0.000,C 90.000,E1 145.388} C_DIS
LIN {X -0.243,Y -494.444,Z 835.603,A 0.000,B 0.000,C 90.000,E1 144.482} C_DIS
LIN {X 0.164,Y -498.716,Z 835.599,A 0.000,B 0.000,C 90.000,E1 143.829} C_DIS
LIN {X 0.195,Y -504.649,Z 835.594,A 0.000,B 0.000,C 90.000,E1 142.924} C_DIS
LIN {X -0.020,Y -508.540,Z 835.591,A 0.000,B 0.000,C 90.000,E1 142.351} C_DIS
LIN {X -0.119,Y -510.515,Z 835.589,A 0.000,B 0.000,C 90.000,E1 142.065} C_DIS
LIN {X -0.177,Y -514.944,Z 835.585,A 0.000,B 0.000,C 90.000,E1 141.331} C_DIS
LIN {X 0.073,Y -521.033,Z 835.579,A 0.000,B 0.000,C 90.000,E1 140.275} C_DIS
LIN {X 0.113,Y -525.089,Z 835.575,A 0.000,B 0.000,C 90.000,E1 139.542} C_DIS
LIN {X -0.214,Y -529.052,Z 835.571,A 0.000,B 0.000,C 90.000,E1 138.852} C_DIS
LIN {X 0.080,Y -532.165,Z 835.568,A 0.000,B 0.000,C 90.000,E1 138.243} C_DIS
LIN {X 0.131,Y -540.239,Z 835.559,A 0.000,B 0.000,C 90.000,E1 136.662} C_DIS
LIN {X -0.053,Y -546.861,Z 835.552,A 0.000,B 0.000,C 90.000,E1 135.405} C_DIS
LIN {X 0.038,Y -552.652,Z 835.546,A 0.000,B 0.000,C 90.000,E1 134.271} C_DIS
LIN {X 0.114,Y -555.412,Z 835.543,A 0.000,B 0.000,C 90.000,E1 133.704} C_DIS
LIN {X 0.168,Y -561.176,Z 835.536,A 0.000,B 0.000,C 90.000,E1 132.447} C_DIS
LIN {X 0.042,Y -567.902,Z 835.528,A 0.000,B 0.000,C 90.000,E1 130.943} C_DIS
LIN {X 0.156,Y -573.621,Z 835.520,A 0.000,B 0.000,C 90.000,E1 129.564} C_DIS
LIN {X -0.013,Y -578.618,Z 835.512,A 0.000,B 0.000,C 90.000,E1 128.222} C_DIS
LIN {X -0.342,Y -581.330,Z 835.508,A 0.000,B 0.000,C 90.000,E1 127.443} C_DIS
LIN {X 0.357,Y -584.296,Z 835.502,A 0.000,B 0.000,C 90.000,E1 126.297} C_DIS
LIN {X 0.092,Y -586.239,Z 835.497,A 0.000,B 0.000,C 90.000,E1 125.518} C_DIS
LIN {X 0.036,Y -588.459,Z 835.491,A 0.000,B 0.000,C 90.000,E1 124.452} C_DIS
LIN {X -0.033,Y -589.825,Z 835.487,A 0.000,B 0.000,C 90.000,E1 123.658} C_DIS
LIN {X -0.170,Y -591.603,Z 835.480,A 0.000,B 0.000,C 90.000,E1 122.339} C_DIS
LIN {X -0.193,Y -592.420,Z 835.475,A 0.000,B 0.000,C 90.000,E1 121.544} C_DIS
LIN {X 0.102,Y -592.892,Z 835.471,A 0.000,B 0.000,C 90.000,E1 120.718} C_DIS
LIN {X 0.093,Y -593.139,Z 835.466,A 0.000,B 0.000,C 90.000,E1 119.922} C_DIS
LIN {X -0.106,Y -593.194,Z 835.463,A 0.000,B 0.000,C 90.000,E1 119.411} C_DIS
LIN {X -0.111,Y -592.925,Z 835.459,A 0.000,B 0.000,C 90.000,E1 118.615} C_DIS
LIN {X 0.301,Y -592.343,Z 835.453,A 0.000,B 0.000,C 90.000,E1 117.513} C_DIS
LIN {X 0.006,Y -591.641,Z 835.449,A 0.000,B 0.000,C 90.000,E1 116.744} C_DIS
LIN {X 0.136,Y -590.250,Z 835.443,A 0.000,B 0.000,C 90.000,E1 115.668} C_DIS
LIN {X -0.071,Y -589.305,Z 835.440,A 0.000,B 0.000,C 90.000,E1 115.155} C_DIS
LIN {X 0.137,Y -587.748,Z 835.435,A 0.000,B 0.000,C 90.000,E1 114.335} C_DIS
LIN {X -0.092,Y -586.092,Z 835.432,A 0.000,B 0.000,C 90.000,E1 113.823} C_DIS
LIN {X 0.325,Y -585.100,Z 835.431,A 0.000,B 0.000,C 90.000,E1 113.515} C_DIS
LIN {X -0.152,Y -582.657,Z 835.428,A 0.000,B 0.000,C 90.000,E1 113.025} C_DIS
LIN {X 0.184,Y -580.483,Z 835.426,A 0.000,B 0.000,C 90.000,E1 112.589} C_DIS
LIN {X 0.115,Y -579.355,Z 835.425,A 0.000,B 0.000,C 90.000,E1 112.461} C_DIS
LIN {X -0.058,Y -575.336,Z 835.423,A 0.000,B 0.000,C 90.000,E1 112.078} C_DIS
LIN {X -0.154,Y -572.048,Z 835.421,A 0.000,B 0.000,C 90.000,E1 111.844} C_DIS
LIN {X -0.074,Y -568.712,Z 835.420,A 0.000,B 0.000,C 90.000,E1 111.535} C_DIS
LIN {X -0.023,Y -567.070,Z 835.419,A 0.000,B 0.000,C 90.000,E1 111.408} C_DIS
LIN {X -0.107,Y -565.639,Z 835.418,A 0.000,B 0.000,C 90.000,E1 111.227} C_DIS
LIN {X 0.128,Y -564.395,Z 835.416,A 0.000,B 0.000,C 90.000,E1 110.791} C_DIS
LIN {X 0.277,Y -564.117,Z 835.414,A 0.000,B 0.000,C 90.000,E1 110.429} C_DIS
LIN {X 0.073,Y -563.537,Z 835.412,A 0.000,B 0.000,C 90.000,E1 110.174} C_DIS
LIN {X 0.204,Y -563.299,Z 835.411,A 0.000,B 0.000,C 90.000,E1 109.885} C_DIS
LIN {X 0.035,Y -562.442,Z 835.406,A 0.000,B 0.000,C 90.000,E1 109.087} C_DIS
LIN {X 0.176,Y -561.903,Z 835.398,A 0.000,B 0.000,C 90.000,E1 107.692} C_DIS
LIN {X -0.244,Y -562.628,Z 835.375,A 0.000,B 0.000,C 90.000,E1 103.592} C_DIS
LIN {X -0.063,Y -563.937,Z 835.363,A 0.000,B 0.000,C 90.000,E1 101.366} C_DIS
LIN {X 0.053,Y -565.495,Z 835.351,A 0.000,B 0.000,C 90.000,E1 99.151} C_DIS
LIN {X 0.246,Y -566.425,Z 835.343,A 0.000,B 0.000,C 90.000,E1 97.757} C_DIS
LIN {X -0.090,Y -567.436,Z 835.334,A 0.000,B 0.000,C 90.000,E1 96.144} C_DIS
LIN {X 0.049,Y -568.117,Z 835.327,A 0.000,B 0.000,C 90.000,E1 94.759} C_DIS
LIN {X 0.256,Y -568.770,Z 835.317,A 0.000,B 0.000,C 90.000,E1 93.094} C_DIS
